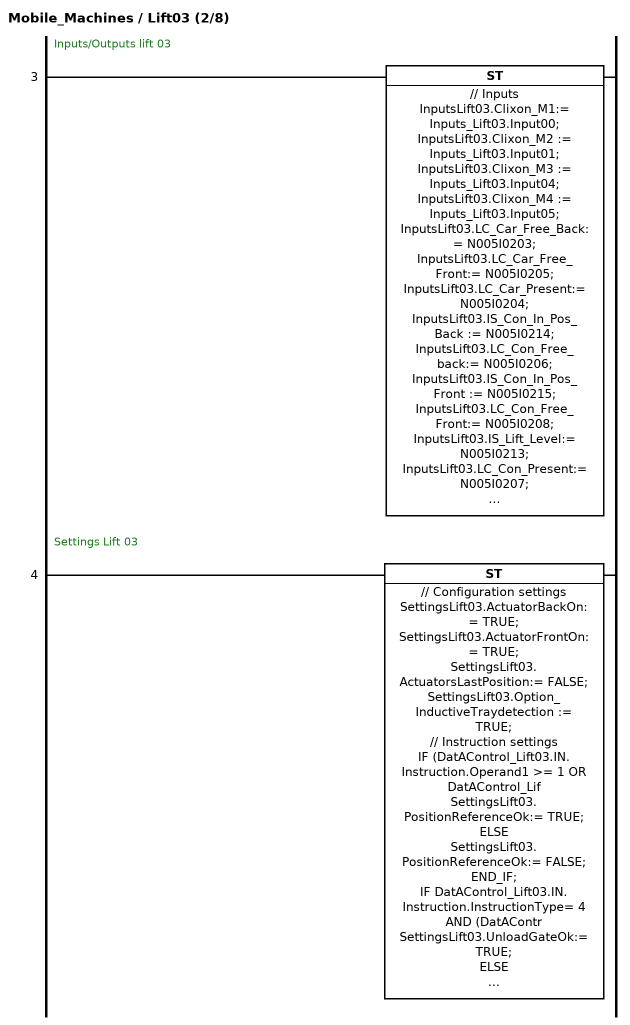
(* [picture p6: Mobile_Machines / Lift03, rungs 3-4] *)
(* Rung 3: Inputs/Outputs lift 03 *)
// Inputs
InputsLift03.Clixon_M1:= Inputs_Lift03.Input00;
InputsLift03.Clixon_M2 := Inputs_Lift03.Input01;
InputsLift03.Clixon_M3 := Inputs_Lift03.Input04;
InputsLift03.Clixon_M4 := Inputs_Lift03.Input05;
InputsLift03.LC_Car_Free_Back:= N005I0203;
InputsLift03.LC_Car_Free_Front:= N005I0205;
InputsLift03.LC_Car_Present:= N005I0204;
InputsLift03.IS_Con_In_Pos_Back := N005I0214;
InputsLift03.LC_Con_Free_back:= N005I0206;
InputsLift03.IS_Con_In_Pos_Front := N005I0215;
InputsLift03.LC_Con_Free_Front:= N005I0208;
InputsLift03.IS_Lift_Level:= N005I0213;
InputsLift03.LC_Con_Present:= N005I0207;
InputsLift03.LS_FallProtect:= N005I0200 OR TRUE;
InputsLift03.LS_Lift_Down:= N005I0202;
InputsLift03.LS_Lift_Up:= N005I0201;
InputsLift03.IS_Act_Back_In:= N005I0210; // Stopper blocks carrier
InputsLift03.IS_Act_Back_Out:= N005I0209; // Carrier can drive in
InputsLift03.IS_Act_Front_In:= N005I0212; // Stopper blocks carrier
InputsLift03.IS_Act_Front_Out:= N005I0211; // Carrier can drive in
InputsLift03.RC_Tray_Stopper_Min_Back_Up:= Inputs_Lift03_Ch.Input00;
InputsLift03.RC_Tray_Stopper_Max_Back_Up:= Inputs_Lift03_Ch.Input01;
InputsLift03.RC_Tray_Stopper_Min_Front_Up:= Inputs_Lift03_Ch.Input04;
InputsLift03.RC_Tray_Stopper_Max_Front_Up:= Inputs_Lift03_Ch.Input05;
InputsLift03.IO_OK := FALSE;
IF NOT N05_Major_Fault AND NOT N05_Minor_Fault AND NOT N05_Partial_Fault AND NOT N33_Major_Fault AND NOT N33_Minor_Fault AND NOT N33_Partial_Fault THEN
 InputsLift03.IO_OK := TRUE;
END_IF;

// Inputs rack
InputsLift03.LC_Lift_Free_Back[0]:= N005I0300;
InputsLift03.LC_Lift_Free_Back[1]:= TRUE;
InputsLift03.LC_Lift_Free_Back[2]:= TRUE;
InputsLift03.LC_Lift_Free_Back[3]:= TRUE;
InputsLift03.LC_Lift_Free_Back[4]:= N005I0304;
InputsLift03.LC_Lift_Free_Back[5]:= TRUE;
InputsLift03.LC_Lift_Free_Back[6]:= TRUE;
InputsLift03.LC_Lift_Free_Back[7]:= TRUE;
InputsLift03.LC_Lift_Free_Back[8]:= TRUE;
InputsLift03.LC_Lift_Free_Back[9]:= TRUE;
InputsLift03.LC_Lift_Free_Back[10]:= TRUE;
InputsLift03.LC_Lift_Free_Back[11]:= TRUE;
InputsLift03.LC_Lift_Free_Back[12]:= TRUE;
InputsLift03.LC_Lift_Free_Back[13]:= TRUE;
InputsLift03.LC_Lift_Free_Back[14]:= TRUE;
InputsLift03.LC_Lift_Free_Back[15]:= TRUE;

InputsLift03.LC_Lift_Free_Front[0]:= N005I0308;
InputsLift03.LC_Lift_Free_Front[1]:= N005I0309;
InputsLift03.LC_Lift_Free_Front[2]:= N005I0310;
InputsLift03.LC_Lift_Free_Front[3]:= N005I0311;
InputsLift03.LC_Lift_Free_Front[4]:= N005I0312;
InputsLift03.LC_Lift_Free_Front[5]:= N005I0313;
InputsLift03.LC_Lift_Free_Front[6]:= N005I0314;
InputsLift03.LC_Lift_Free_Front[7]:= N005I0315;
InputsLift03.LC_Lift_Free_Front[8]:= TRUE;
InputsLift03.LC_Lift_Free_Front[9]:= TRUE;
InputsLift03.LC_Lift_Free_Front[10]:= TRUE;
InputsLift03.LC_Lift_Free_Front[11]:= TRUE;
InputsLift03.LC_Lift_Free_Front[12]:= TRUE;
InputsLift03.LC_Lift_Free_Front[13]:= TRUE;
InputsLift03.LC_Lift_Free_Front[14]:= TRUE;
InputsLift03.LC_Lift_Free_Front[15]:= TRUE;

// Martins inputs
Lift03_SafetyInput1 := Inputs_Lift03.Input02;
Lift03_SafetyInput2 := Inputs_Lift03.Input03;

Knop_FW_Lift03 := N005I0301;
Knop_RV_Lift03 := N005I0302;
Knop_OK_Lift03 := N005I0303;
Knop_Snel_Lift03 := N005I0305;

// Outputs
N005O400:= OutputsLift03.Brake_Back;
// N005O401:= OutputsLift03.Actuator_Back_Out;
// N005O402:= OutputsLift03.Actuator_Back_In;
N005O403:= OutputsLift03.Actuator_Front_Out;
N005O404:= OutputsLift03.Actuator_Front_In;
N005O405 := OutputsLift03.Brake_Front; // Pls use only hold the brake and not release it for a correction
N005O406 := Led_RS_Extern;
N005O407 := OutputsLift03.V_TrayStopper_Front_Up;
LiftGR03NotLoaded := OutputsLift03.LC_Container_Free;

Comm_To_Carrier01.Lift_Info.CarrierNot_Loaded_Lift1 := FALSE; 
Comm_To_Carrier02.Lift_Info.CarrierNot_Loaded_Lift1 := FALSE;
Comm_To_Carrier03.Lift_Info.CarrierNot_Loaded_Lift1 := FALSE;
Comm_To_Carrier04.Lift_Info.CarrierNot_Loaded_Lift1 := FALSE;
Comm_To_Carrier05.Lift_Info.CarrierNot_Loaded_Lift1 := FALSE;

IF OutputsLift03.LC_Carrier_Free THEN
Comm_To_Carrier01.Lift_Info.CarrierNot_Loaded_Lift1 := TRUE; 
Comm_To_Carrier02.Lift_Info.CarrierNot_Loaded_Lift1 := TRUE;
Comm_To_Carrier03.Lift_Info.CarrierNot_Loaded_Lift1 := TRUE;
Comm_To_Carrier04.Lift_Info.CarrierNot_Loaded_Lift1 := TRUE;
Comm_To_Carrier05.Lift_Info.CarrierNot_Loaded_Lift1 := TRUE;
END_IF;

Comm_To_Carrier01.Lift_Info.TrayNot_Loaded_Lift1 := FALSE;
Comm_To_Carrier02.Lift_Info.TrayNot_Loaded_Lift1 := FALSE;
Comm_To_Carrier03.Lift_Info.TrayNot_Loaded_Lift1 := FALSE;
Comm_To_Carrier04.Lift_Info.TrayNot_Loaded_Lift1 := FALSE;
Comm_To_Carrier05.Lift_Info.TrayNot_Loaded_Lift1 := FALSE;

IF OutputsLift03.LC_Container_Free THEN
Comm_To_Carrier01.Lift_Info.TrayNot_Loaded_Lift1 := TRUE;
Comm_To_Carrier02.Lift_Info.TrayNot_Loaded_Lift1 := TRUE;
Comm_To_Carrier03.Lift_Info.TrayNot_Loaded_Lift1 := TRUE;
Comm_To_Carrier04.Lift_Info.TrayNot_Loaded_Lift1 := TRUE;
Comm_To_Carrier05.Lift_Info.TrayNot_Loaded_Lift1 := TRUE;
END_IF;
(* Rung 4: Settings Lift 03 *)
// Configuration settings
SettingsLift03.ActuatorBackOn:= TRUE;
SettingsLift03.ActuatorFrontOn:= TRUE;
SettingsLift03.ActuatorsLastPosition:= FALSE;
SettingsLift03.Option_InductiveTraydetection := TRUE;

// Instruction settings
IF (DatAControl_Lift03.IN.Instruction.Operand1 >= 1 OR DatAControl_Lift03.IN.Instruction.Operand1 <= 7) THEN
	SettingsLift03.PositionReferenceOk:= TRUE;
ELSE
	SettingsLift03.PositionReferenceOk:= FALSE;
END_IF;

IF DatAControl_Lift03.IN.Instruction.InstructionType= 4 AND (DatAControl_Lift03.IN.Instruction.Operand1 = 102 OR DatAControl_Lift03.IN.Instruction.Operand1 = 602) THEN
	SettingsLift03.UnloadGateOk:= TRUE;
ELSE
	SettingsLift03.UnloadGateOk:=FALSE;
END_IF;

IF DatAControl_Lift03.IN.Instruction.InstructionType= 3 AND (DatAControl_Lift03.IN.Instruction.Operand1 = 102 OR DatAControl_Lift03.IN.Instruction.Operand1 = 602) THEN
	SettingsLift03.LoadGateOk:= TRUE;
ELSE
	SettingsLift03.LoadGateOk:= FALSE;
END_IF;

// Parameters
SettingsLift03.MachineCode:=4;
SettingsLift03.SafeStopTime:=15;
SettingsLift03.Tolerance_At_Position:=50;
SettingsLift03.Warning_Tolerance_At_Position:=25;
SettingsLift03.BrakeReleaseFreq:=750;
SettingsLift03.Dec_Area_High:= 10000;
SettingsLift03.Dec_Area_Low:=1000;
SettingsLift03.NodeNummerLift:=9;
SettingsLift03.NodeNummerChain:=10;
SettingsLift03.MinimumSpeed:=1000;
SettingsLift03.MaximumSpeed:=8400; // Motor with extern brake 84Hz max, motor with no brake 87Hz max
SettingsLift03.MinimumSpeedChain:= 3700;
SettingsLift03.MaximumSpeedChain:= 8000; // Motor with intern brake 68 Hz max
SettingsLift03.TimeConFreeBackDOFF:= 50;
SettingsLift03.TimeConFreeBackDON:= 5;
SettingsLift03.TimeConFreeFrontDOFF:= 5;
SettingsLift03.TimeConFreeFrontDON:= 5;
SettingsLift03.UseBenchUnloadInstruction:= TRUE;

IF Commands_Lift03.Reverse THEN // Slow down
	SettingsLift03.MinimumSpeed := 750;
	SettingsLift03.BrakeReleaseFreq:=500;
END_IF;

IF SettingsLift03.Option_InductiveTraydetection THEN
	SettingsLift03.ChainHighSpeed := 60;
ELSE
 	SettingsLift03.ChainHighSpeed := 85;
END_IF;

SettingsLift03.TimeConInductiveBackDOFF := 2;
SettingsLift03.TimeConInductiveBackDON := 8;
SettingsLift03.TimeConInductiveFrontDOFF := 2;
SettingsLift03.TimeConInductiveFrontDON := 8;

// Mechanical settings 1mm = 17 pulses
SettingsLift03.MinimumPulseLevel:=10000;
SettingsLift03.MaximumPulseLevel:=177000;
SettingsLift03.TooFarAllowed:= 1000;
SettingsLift03.ResetValueMargin := 500;
SettingsLift03.MinimumPosition:= 1;
SettingsLift03.MaximumPosition:= 9;
SettingsLift03.PulseLevel[1]:=10000;
SettingsLift03.PulseLevel[2]:= Lift3_PulsValueLevel2; // 13345;
SettingsLift03.PulseLevel[3]:= Lift3_PulsValueLevel3; // 49853 // 49790
SettingsLift03.PulseLevel[4]:= Lift3_PulsValueLevel4; // 70329 // 70240; 
SettingsLift03.PulseLevel[5]:= Lift3_PulsValueLevel5; // 90761 // 90690; 
SettingsLift03.PulseLevel[6]:= Lift3_PulsValueLevel6; // 111397 // 111140; 
SettingsLift03.PulseLevel[7]:= Lift3_PulsValueLevel7; // 131690 // 131590;
SettingsLift03.PulseLevel[8]:= Lift3_PulsValueLevel8; // 152156 // 152040; 
SettingsLift03.PulseLevel[9]:= Lift3_PulsValueLevel9; // 172626 // 172490; 
SettingsLift03.PulseLevel[10]:=10;
SettingsLift03.PulseLevel[11]:=10;
SettingsLift03.PulseLevel[12]:=10;
SettingsLift03.PulseLevel[13]:=10;
SettingsLift03.PulseLevel[14]:=10;
SettingsLift03.PulseLevel[15]:=10;

SettingsLift03.NeedLevelSensor[1]:=FALSE;
SettingsLift03.NeedLevelSensor[2]:=FALSE;
SettingsLift03.NeedLevelSensor[3]:=TRUE;
SettingsLift03.NeedLevelSensor[4]:=TRUE;
SettingsLift03.NeedLevelSensor[5]:=TRUE;
SettingsLift03.NeedLevelSensor[6]:=TRUE;
SettingsLift03.NeedLevelSensor[7]:=TRUE;
SettingsLift03.NeedLevelSensor[8]:=TRUE;
SettingsLift03.NeedLevelSensor[9]:=TRUE;
SettingsLift03.NeedLevelSensor[10]:=TRUE;
SettingsLift03.NeedLevelSensor[11]:=TRUE;
SettingsLift03.NeedLevelSensor[12]:=TRUE;
SettingsLift03.NeedLevelSensor[13]:=TRUE;
SettingsLift03.NeedLevelSensor[14]:=TRUE;
SettingsLift03.NeedLevelSensor[15]:=TRUE;

// SettingsLift03.BrakeReleaseFreq:=750; SettingsLift03.MinimumSpeed:=1000;
// When rev setting: SettingsLift03.MinimumSpeed := 750; SettingsLift03.BrakeReleaseFreq:=500;
// Acc 20sec, dec 4sec

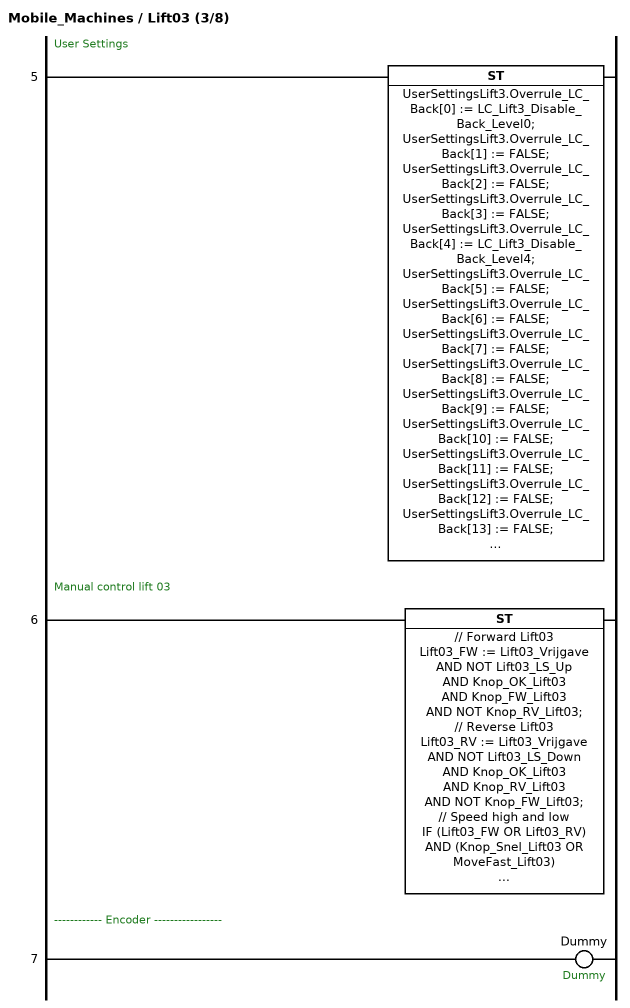
(* Rung 5: User Settings *)
UserSettingsLift3.Overrule_LC_Back[0] := LC_Lift3_Disable_Back_Level0;
UserSettingsLift3.Overrule_LC_Back[1] := FALSE;
UserSettingsLift3.Overrule_LC_Back[2] := FALSE;
UserSettingsLift3.Overrule_LC_Back[3] := FALSE;
UserSettingsLift3.Overrule_LC_Back[4] := LC_Lift3_Disable_Back_Level4;
UserSettingsLift3.Overrule_LC_Back[5] := FALSE;
UserSettingsLift3.Overrule_LC_Back[6] := FALSE;
UserSettingsLift3.Overrule_LC_Back[7] := FALSE;
UserSettingsLift3.Overrule_LC_Back[8] := FALSE;
UserSettingsLift3.Overrule_LC_Back[9] := FALSE;
UserSettingsLift3.Overrule_LC_Back[10] := FALSE;
UserSettingsLift3.Overrule_LC_Back[11] := FALSE;
UserSettingsLift3.Overrule_LC_Back[12] := FALSE;
UserSettingsLift3.Overrule_LC_Back[13] := FALSE;
UserSettingsLift3.Overrule_LC_Back[14] := FALSE;
UserSettingsLift3.Overrule_LC_Back[15] := FALSE;

UserSettingsLift3.Overrule_LC_Front[0] := LC_Lift3_Disable_Front_Level0;
UserSettingsLift3.Overrule_LC_Front[1] := LC_Lift3_Disable_Front_Level1;
UserSettingsLift3.Overrule_LC_Front[2] := LC_Lift3_Disable_Front_Level2;
UserSettingsLift3.Overrule_LC_Front[3] := LC_Lift3_Disable_Front_Level3;
UserSettingsLift3.Overrule_LC_Front[4] := LC_Lift3_Disable_Front_Level4;
UserSettingsLift3.Overrule_LC_Front[5] := LC_Lift3_Disable_Front_Level5;
UserSettingsLift3.Overrule_LC_Front[6] := LC_Lift3_Disable_Front_Level6;
UserSettingsLift3.Overrule_LC_Front[7] := LC_Lift3_Disable_Front_Level7;
UserSettingsLift3.Overrule_LC_Front[8] := FALSE;
UserSettingsLift3.Overrule_LC_Front[9] := FALSE;
UserSettingsLift3.Overrule_LC_Front[10] := FALSE;
UserSettingsLift3.Overrule_LC_Front[11] := FALSE;
UserSettingsLift3.Overrule_LC_Front[12] := FALSE;
UserSettingsLift3.Overrule_LC_Front[13] := FALSE;
UserSettingsLift3.Overrule_LC_Front[14] := FALSE;
UserSettingsLift3.Overrule_LC_Front[15] := FALSE;
(* Rung 6: Manual control lift 03 *)
// Forward Lift03
Lift03_FW := Lift03_Vrijgave
AND NOT Lift03_LS_Up
AND Knop_OK_Lift03
AND Knop_FW_Lift03
AND NOT Knop_RV_Lift03;
// Reverse Lift03
Lift03_RV := Lift03_Vrijgave
AND NOT Lift03_LS_Down
AND Knop_OK_Lift03
AND Knop_RV_Lift03
AND NOT Knop_FW_Lift03;

// Speed high and low
IF (Lift03_FW OR Lift03_RV) AND (Knop_Snel_Lift03 OR MoveFast_Lift03)
AND EncoderLift03>SettingsLift03.MinimumPulseLevel+1000 AND EncoderLift03<SettingsLift03.MaximumPulseLevel-1000 THEN
	SettingsLift03.MinimumSpeed:=5000;
END_IF;

// Led ok Lift03
Led_Knop_OK_Lift03 := Knop_OK_Lift03 AND Lift03_Vrijgave;

// Vrijgave Lift03
Lift03_Vrijgave := (*Lift03_LS_FallProtect
AND*) Lift03_SafetyInput1 AND Lift03_SafetyInput2 AND Lift03_Alarms=0;

// Use manual control buttons as replacement for pocket (TEMP)
//Lift03_FW  Lift03_RV
IF Knop_OK_Lift03 THEN
	Pocket_Lift03.Move.Out:=Lift03_FW;
	Pocket_Lift03.Move.In:= Lift03_RV;
	Pocket_Lift03.Move.Stop:= NOT Lift03_FW AND NOT Lift03_RV;
END_IF;

// Move fast on/off
IF Pocket_Lift03.MoveFastOn THEN
	MoveFast_Lift03 := TRUE;
END_IF;
IF Pocket_Lift03.MoveFastOff OR DatAControl_Lift03.IN.MachineMode<>3 THEN
	MoveFast_Lift03 := FALSE;
END_IF;
Pocket_Lift03.MoveFastOn := FALSE;
Pocket_Lift03.MoveFastOff := FALSE;
(* Rung 7: ------------ Encoder ----------------- *)
Dummy := TRUE;

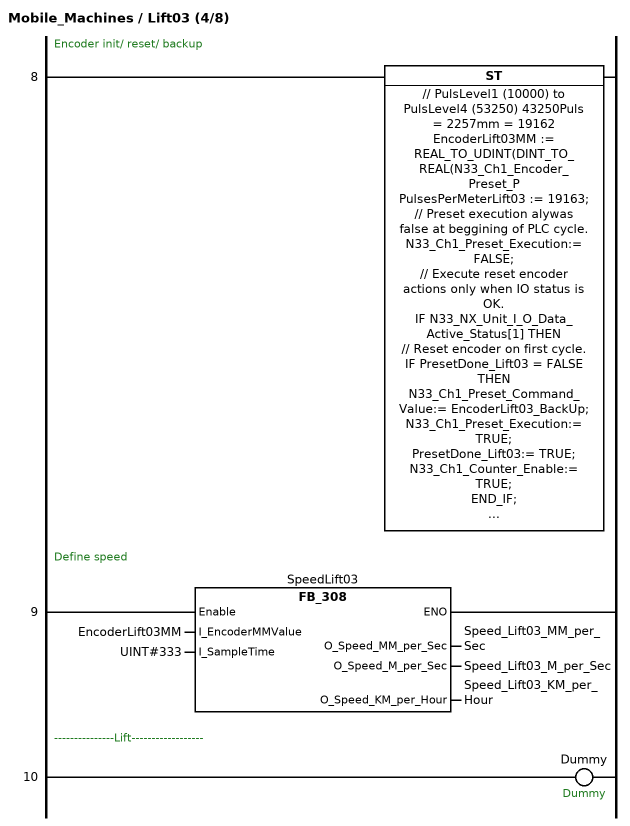
(* Rung 8: Encoder init/ reset/ backup *)
// PulsLevel1 (10000) to PulsLevel4 (53250) 43250Puls = 2257mm = 19162,605228179 PpM
EncoderLift03MM := REAL_TO_UDINT(DINT_TO_REAL(N33_Ch1_Encoder_Preset_Position) / UDINT_TO_REAL(PulsesPerMeterLift03) * 1000);
PulsesPerMeterLift03 := 19163;

// Preset execution alywas false at beggining of PLC cycle.
N33_Ch1_Preset_Execution:= FALSE;

// Execute reset encoder actions only when IO status is OK.
IF N33_NX_Unit_I_O_Data_Active_Status[1] THEN
	
	// Reset encoder on first cycle.
	IF PresetDone_Lift03 = FALSE THEN
		N33_Ch1_Preset_Command_Value:= EncoderLift03_BackUp;
		N33_Ch1_Preset_Execution:= TRUE;
		PresetDone_Lift03:= TRUE;
		N33_Ch1_Counter_Enable:= TRUE;
	END_IF;
	
	// Reset encoder when lift is at position.
	IF ResetEncoder_Lift03 THEN
		N33_Ch1_Preset_Command_Value:= ResetEncoderValue_Lift03; // 10000 @Ground
		N33_Ch1_Preset_Execution:= TRUE;
		ResetEncoder_Lift03:= FALSE;
	END_IF;
	
	// Move encoder value.
    EncoderLift03 := DINT_TO_UDINT(N33_Ch1_Encoder_Preset_Position);
		
	// Backup encoder value.
	EncoderLift03_Backup:= EncoderLift03;
END_IF;
(* Rung 9: Define speed *)
SpeedLift03(Enable := TRUE, I_EncoderMMValue := EncoderLift03MM, I_SampleTime := UINT#333, O_Speed_MM_per_Sec => Speed_Lift03_MM_per_Sec, O_Speed_M_per_Sec => Speed_Lift03_M_per_Sec, O_Speed_KM_per_Hour => Speed_Lift03_KM_per_Hour);
(* Rung 10: ---------------Lift------------------ *)
Dummy := TRUE;

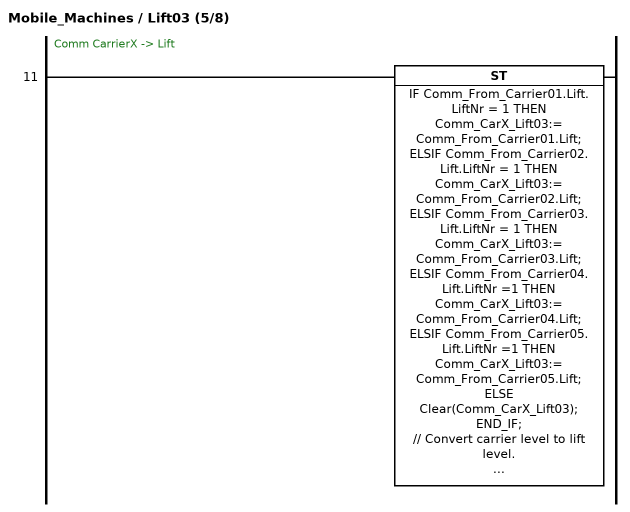
(* Rung 11: Comm CarrierX -> Lift *)
IF Comm_From_Carrier01.Lift.LiftNr = 1 THEN
	Comm_CarX_Lift03:= Comm_From_Carrier01.Lift;
ELSIF Comm_From_Carrier02.Lift.LiftNr = 1 THEN
	Comm_CarX_Lift03:= Comm_From_Carrier02.Lift;
ELSIF Comm_From_Carrier03.Lift.LiftNr = 1 THEN
	Comm_CarX_Lift03:= Comm_From_Carrier03.Lift;
ELSIF Comm_From_Carrier04.Lift.LiftNr =1 THEN
	Comm_CarX_Lift03:= Comm_From_Carrier04.Lift;
ELSIF Comm_From_Carrier05.Lift.LiftNr =1 THEN
	Comm_CarX_Lift03:= Comm_From_Carrier05.Lift;
ELSE
	Clear(Comm_CarX_Lift03);
END_IF;

// Convert carrier level to lift level.
//This is only needed when lift has more levels than the carrier!
CASE Comm_CarX_Lift03.Height_MobileMachine OF
	1: Comm_CarX_Lift03.Height_MobileMachine:=3;
	2: Comm_CarX_Lift03.Height_MobileMachine:=4;
	// mezzanine will probably add an extra level to the lift ones.
	3: Comm_CarX_Lift03.Height_MobileMachine:=5;
	4: Comm_CarX_Lift03.Height_MobileMachine:=6;
	5: Comm_CarX_Lift03.Height_MobileMachine:=7;
	6: Comm_CarX_Lift03.Height_MobileMachine:=8;
	7: Comm_CarX_Lift03.Height_MobileMachine:=9;
ELSE
	// If lift drops the carrier on a level not listed above set to 0 to avoid wrong positions.
     Comm_CarX_Lift03.Height_MobileMachine:=0;
END_CASE;

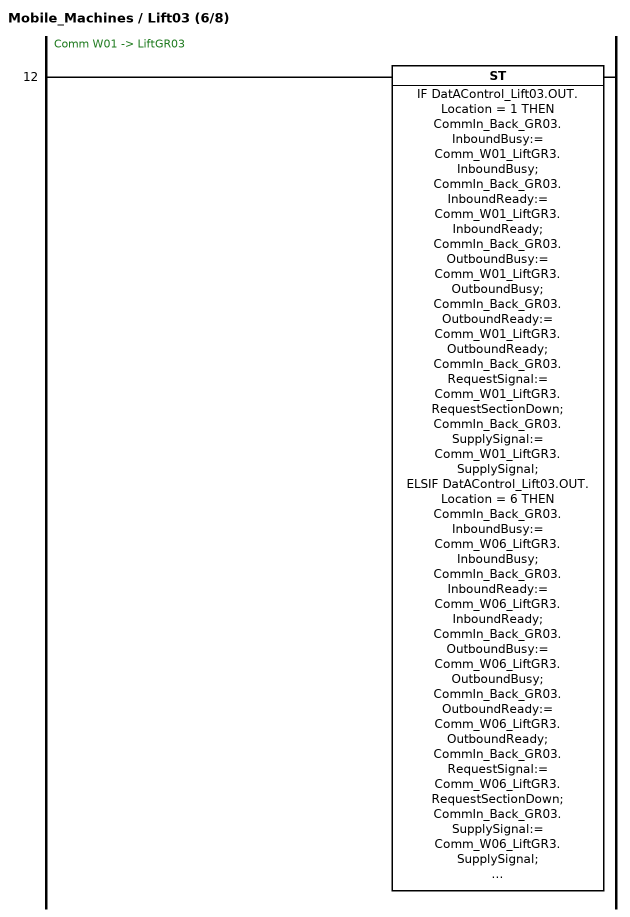
(* Rung 12: Comm W01 -> LiftGR03 *)
IF DatAControl_Lift03.OUT.Location = 1 THEN
CommIn_Back_GR03.InboundBusy:= Comm_W01_LiftGR3.InboundBusy;
CommIn_Back_GR03.InboundReady:= Comm_W01_LiftGR3.InboundReady;
CommIn_Back_GR03.OutboundBusy:= Comm_W01_LiftGR3.OutboundBusy;
CommIn_Back_GR03.OutboundReady:= Comm_W01_LiftGR3.OutboundReady;
CommIn_Back_GR03.RequestSignal:= Comm_W01_LiftGR3.RequestSectionDown;
CommIn_Back_GR03.SupplySignal:= Comm_W01_LiftGR3.SupplySignal;
ELSIF DatAControl_Lift03.OUT.Location = 6 THEN
CommIn_Back_GR03.InboundBusy:= Comm_W06_LiftGR3.InboundBusy;
CommIn_Back_GR03.InboundReady:= Comm_W06_LiftGR3.InboundReady;
CommIn_Back_GR03.OutboundBusy:= Comm_W06_LiftGR3.OutboundBusy;
CommIn_Back_GR03.OutboundReady:= Comm_W06_LiftGR3.OutboundReady;
CommIn_Back_GR03.RequestSignal:= Comm_W06_LiftGR3.RequestSectionDown;
CommIn_Back_GR03.SupplySignal:= Comm_W06_LiftGR3.SupplySignal;
END_IF;

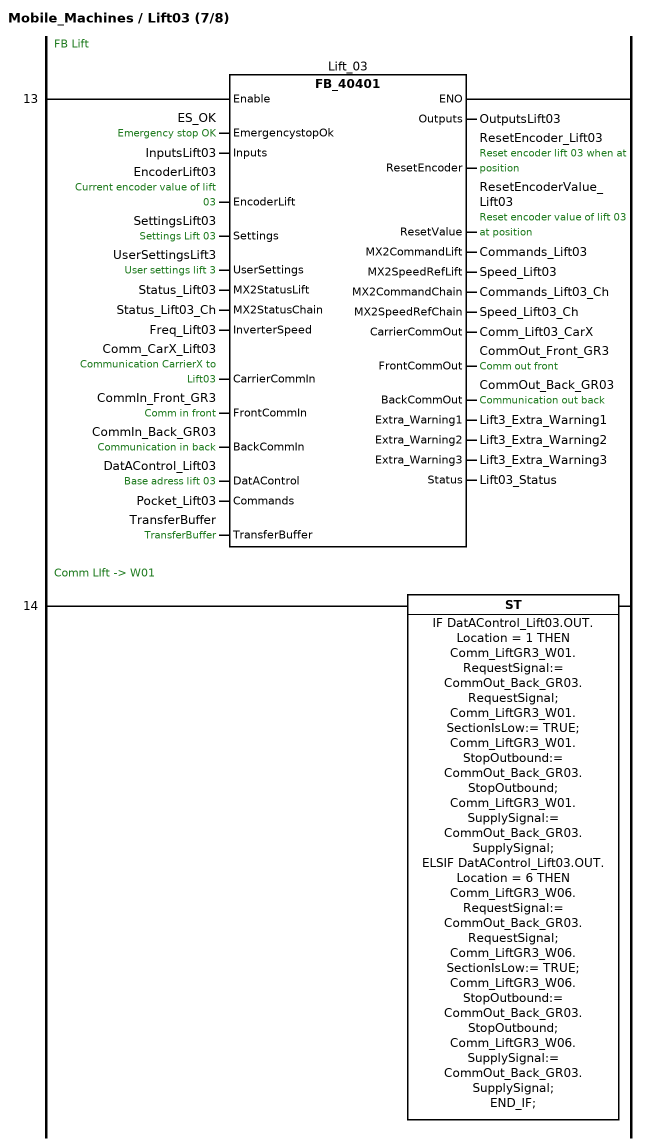
(* Rung 13: FB Lift *)
Lift_03(Enable := TRUE, EmergencystopOk := ES_OK, Inputs := InputsLift03, EncoderLift := EncoderLift03, Settings := SettingsLift03, UserSettings := UserSettingsLift3, MX2StatusLift := Status_Lift03, MX2StatusChain := Status_Lift03_Ch, InverterSpeed := Freq_Lift03, CarrierCommIn := Comm_CarX_Lift03, FrontCommIn := CommIn_Front_GR3, BackCommIn := CommIn_Back_GR03, DatAControl := DatAControl_Lift03, Commands := Pocket_Lift03, TransferBuffer := TransferBuffer, Outputs => OutputsLift03, ResetEncoder => ResetEncoder_Lift03, ResetValue => ResetEncoderValue_Lift03, MX2CommandLift => Commands_Lift03, MX2SpeedRefLift => Speed_Lift03, MX2CommandChain => Commands_Lift03_Ch, MX2SpeedRefChain => Speed_Lift03_Ch, CarrierCommOut => Comm_Lift03_CarX, FrontCommOut => CommOut_Front_GR3, BackCommOut => CommOut_Back_GR03, Extra_Warning1 => Lift3_Extra_Warning1, Extra_Warning2 => Lift3_Extra_Warning2, Extra_Warning3 => Lift3_Extra_Warning3, Status => Lift03_Status);
(* Rung 14: Comm LIft -> W01 *)
IF DatAControl_Lift03.OUT.Location = 1 THEN
Comm_LiftGR3_W01.RequestSignal:= CommOut_Back_GR03.RequestSignal;
Comm_LiftGR3_W01.SectionIsLow:= TRUE;
Comm_LiftGR3_W01.StopOutbound:= CommOut_Back_GR03.StopOutbound;
Comm_LiftGR3_W01.SupplySignal:= CommOut_Back_GR03.SupplySignal;
ELSIF DatAControl_Lift03.OUT.Location = 6 THEN
Comm_LiftGR3_W06.RequestSignal:= CommOut_Back_GR03.RequestSignal;
Comm_LiftGR3_W06.SectionIsLow:= TRUE;
Comm_LiftGR3_W06.StopOutbound:= CommOut_Back_GR03.StopOutbound;
Comm_LiftGR3_W06.SupplySignal:= CommOut_Back_GR03.SupplySignal;
END_IF;

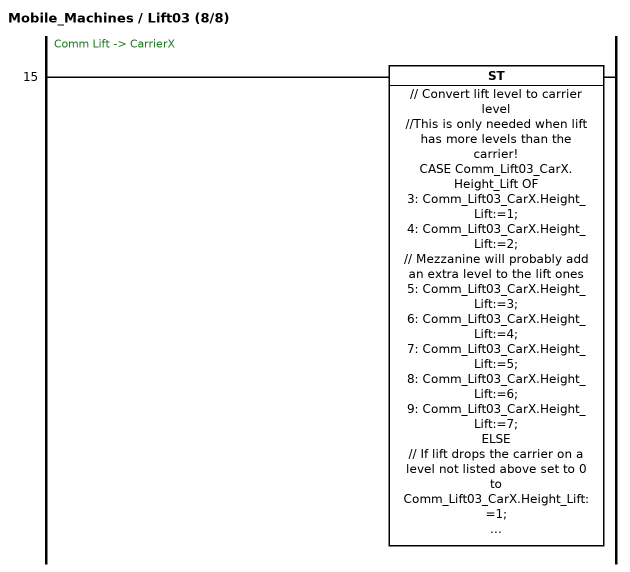
(* Rung 15: Comm Lift -> CarrierX *)
// Convert lift level to carrier level
//This is only needed when lift has more levels than the carrier!
CASE Comm_Lift03_CarX.Height_Lift OF
	3: Comm_Lift03_CarX.Height_Lift:=1;
	4: Comm_Lift03_CarX.Height_Lift:=2;
	// Mezzanine will probably add an extra level to the lift ones
	5: Comm_Lift03_CarX.Height_Lift:=3;
	6: Comm_Lift03_CarX.Height_Lift:=4;
	7: Comm_Lift03_CarX.Height_Lift:=5;
	8: Comm_Lift03_CarX.Height_Lift:=6;
	9: Comm_Lift03_CarX.Height_Lift:=7;
ELSE
	// If lift drops the carrier on a level not listed above set to 0 to avoid wrong positions.
     Comm_Lift03_CarX.Height_Lift:=1;
END_CASE;

IF Comm_From_Carrier01.Lift.LiftNr = 1 THEN
	Comm_To_Carrier01.Lift:= Comm_Lift03_CarX;
ELSIF Comm_From_Carrier02.Lift.LiftNr = 1 THEN
	Comm_To_Carrier02.Lift:= Comm_Lift03_CarX;
ELSIF Comm_From_Carrier03.Lift.LiftNr = 1 THEN
	Comm_To_Carrier03.Lift:= Comm_Lift03_CarX;
ELSIF Comm_From_Carrier04.Lift.LiftNr = 1 THEN
	Comm_To_Carrier04.Lift:= Comm_Lift03_CarX;
ELSIF Comm_From_Carrier05.Lift.LiftNr = 1 THEN
	Comm_To_Carrier05.Lift:= Comm_Lift03_CarX;
END_IF;

(* Section Lift04: ladder, written here as Structured Text *)

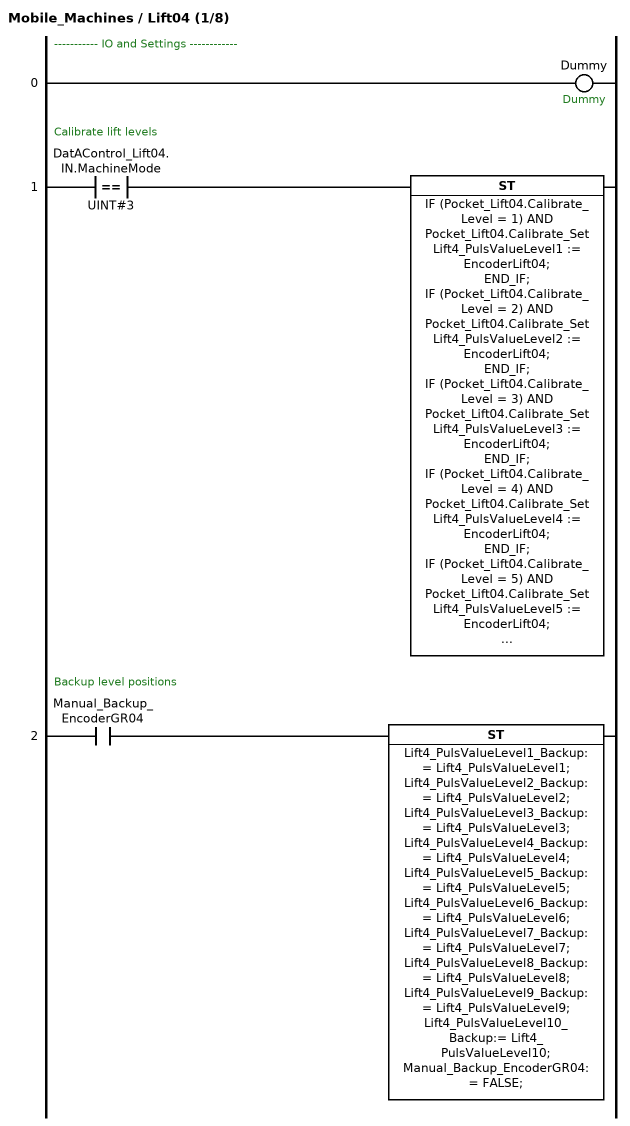
(* Rung 0: ----------- IO and Settings ------------ *)
Dummy := TRUE;
(* Rung 1: Calibrate lift levels *)
IF DatAControl_Lift04.IN.MachineMode = UINT#3 THEN
    IF (Pocket_Lift04.Calibrate_Level = 1) AND Pocket_Lift04.Calibrate_SetLevel THEN
    	Lift4_PulsValueLevel1 := EncoderLift04;
    END_IF;
    
    IF (Pocket_Lift04.Calibrate_Level = 2) AND Pocket_Lift04.Calibrate_SetLevel THEN
    	Lift4_PulsValueLevel2 := EncoderLift04;
    END_IF;
    
    IF (Pocket_Lift04.Calibrate_Level = 3) AND Pocket_Lift04.Calibrate_SetLevel THEN
    	Lift4_PulsValueLevel3 := EncoderLift04;
    END_IF;
    
    IF (Pocket_Lift04.Calibrate_Level = 4) AND Pocket_Lift04.Calibrate_SetLevel THEN
    	Lift4_PulsValueLevel4 := EncoderLift04;
    END_IF;
    
    IF (Pocket_Lift04.Calibrate_Level = 5) AND Pocket_Lift04.Calibrate_SetLevel THEN
    	Lift4_PulsValueLevel5 := EncoderLift04;
    END_IF;
    
    IF (Pocket_Lift04.Calibrate_Level = 6) AND Pocket_Lift04.Calibrate_SetLevel THEN
    	Lift4_PulsValueLevel6 := EncoderLift04;
    END_IF;
    
    IF (Pocket_Lift04.Calibrate_Level = 7) AND Pocket_Lift04.Calibrate_SetLevel THEN
    	Lift4_PulsValueLevel7 := EncoderLift04;
    END_IF;
    
    IF (Pocket_Lift04.Calibrate_Level = 8) AND Pocket_Lift04.Calibrate_SetLevel THEN
    	Lift4_PulsValueLevel8 := EncoderLift04;
    END_IF;
    
    IF (Pocket_Lift04.Calibrate_Level = 9) AND Pocket_Lift04.Calibrate_SetLevel THEN
    	Lift4_PulsValueLevel9 := EncoderLift04;
    END_IF;
    
    IF (Pocket_Lift04.Calibrate_Level = 10) AND Pocket_Lift04.Calibrate_SetLevel THEN
    	Lift4_PulsValueLevel10 := EncoderLift04;
    END_IF;
    
    Pocket_Lift04.Calibrate_SetLevel := FALSE; 
END_IF;
(* Rung 2: Backup level positions *)
IF Manual_Backup_EncoderGR04 THEN
    Lift4_PulsValueLevel1_Backup:= Lift4_PulsValueLevel1;
    Lift4_PulsValueLevel2_Backup:= Lift4_PulsValueLevel2;
    Lift4_PulsValueLevel3_Backup:= Lift4_PulsValueLevel3;
    Lift4_PulsValueLevel4_Backup:= Lift4_PulsValueLevel4;
    Lift4_PulsValueLevel5_Backup:= Lift4_PulsValueLevel5;
    Lift4_PulsValueLevel6_Backup:= Lift4_PulsValueLevel6;
    Lift4_PulsValueLevel7_Backup:= Lift4_PulsValueLevel7;
    Lift4_PulsValueLevel8_Backup:= Lift4_PulsValueLevel8;
    Lift4_PulsValueLevel9_Backup:= Lift4_PulsValueLevel9;
    Lift4_PulsValueLevel10_Backup:= Lift4_PulsValueLevel10;
    
    Manual_Backup_EncoderGR04:= FALSE;
END_IF;

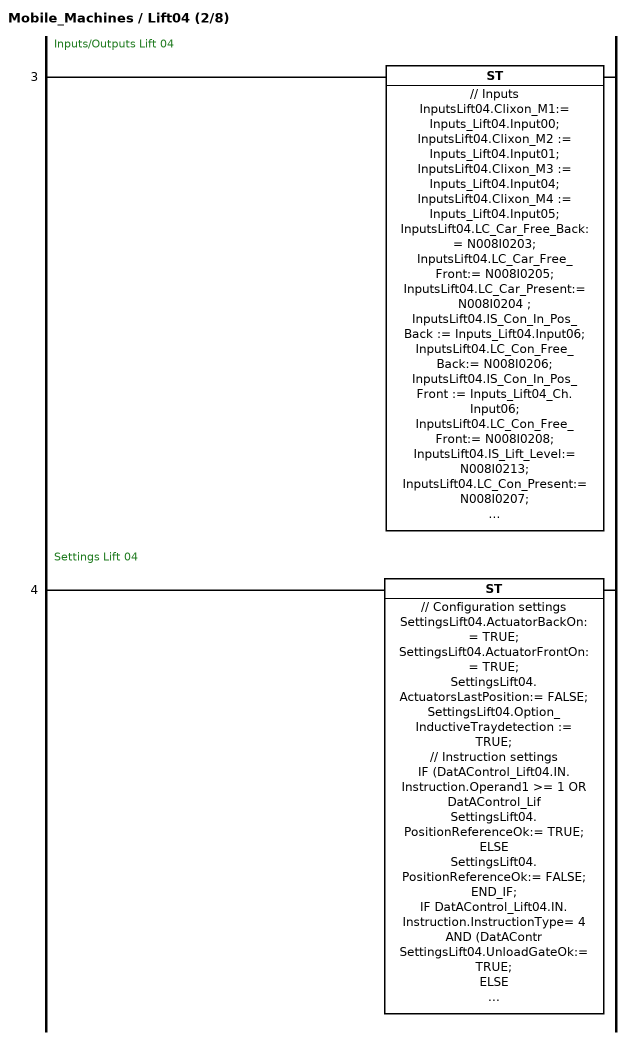
(* Rung 3: Inputs/Outputs Lift 04 *)
// Inputs
InputsLift04.Clixon_M1:= Inputs_Lift04.Input00;
InputsLift04.Clixon_M2 := Inputs_Lift04.Input01;
InputsLift04.Clixon_M3 := Inputs_Lift04.Input04;
InputsLift04.Clixon_M4 := Inputs_Lift04.Input05;
InputsLift04.LC_Car_Free_Back:= N008I0203;
InputsLift04.LC_Car_Free_Front:= N008I0205;
InputsLift04.LC_Car_Present:= N008I0204 ;
InputsLift04.IS_Con_In_Pos_Back := Inputs_Lift04.Input06;
InputsLift04.LC_Con_Free_Back:= N008I0206;
InputsLift04.IS_Con_In_Pos_Front := Inputs_Lift04_Ch.Input06;
InputsLift04.LC_Con_Free_Front:= N008I0208;
InputsLift04.IS_Lift_Level:= N008I0213;
InputsLift04.LC_Con_Present:= N008I0207;
InputsLift04.LS_FallProtect:= N008I0200;
InputsLift04.LS_Lift_Down:= N008I0202;
InputsLift04.LS_Lift_Up:= N008I0201;
InputsLift04.IS_Act_Back_In:= N008I0210; // Stopper blocks carrier
InputsLift04.IS_Act_Back_Out:= N008I0209; // Carrier can drive in
InputsLift04.IS_Act_Front_In:= N008I0212; // Stopper blocks carrier
InputsLift04.IS_Act_Front_Out:= N008I0211; // Carrier can drive in
InputsLift04.RC_Tray_Stopper_Min_Back_Up:= Inputs_Lift04_Ch.Input00;
InputsLift04.RC_Tray_Stopper_Max_Back_Up:= Inputs_Lift04_Ch.Input01;
InputsLift04.RC_Tray_Stopper_Min_Front_Up:= Inputs_Lift04_Ch.Input04;
InputsLift04.RC_Tray_Stopper_Max_Front_Up:= Inputs_Lift04_Ch.Input05;
InputsLift04.IO_OK := FALSE;
IF NOT N08_Major_Fault AND NOT N08_Minor_Fault AND NOT N08_Partial_Fault AND NOT N43_Major_Fault AND NOT N43_Minor_Fault AND NOT N43_Partial_Fault THEN
 InputsLift04.IO_OK := TRUE;
END_IF;

// Inputs rack
InputsLift04.LC_Lift_Free_Back[0]:= N008I0300;
InputsLift04.LC_Lift_Free_Back[1]:= TRUE;
InputsLift04.LC_Lift_Free_Back[2]:= TRUE;
InputsLift04.LC_Lift_Free_Back[3]:= TRUE;
InputsLift04.LC_Lift_Free_Back[4]:= N008I0304;
InputsLift04.LC_Lift_Free_Back[5]:= TRUE;
InputsLift04.LC_Lift_Free_Back[6]:= TRUE;
InputsLift04.LC_Lift_Free_Back[7]:= TRUE;
InputsLift04.LC_Lift_Free_Back[8]:= TRUE;
InputsLift04.LC_Lift_Free_Back[9]:= TRUE;
InputsLift04.LC_Lift_Free_Back[10]:= TRUE;
InputsLift04.LC_Lift_Free_Back[11]:= TRUE;
InputsLift04.LC_Lift_Free_Back[12]:= TRUE;
InputsLift04.LC_Lift_Free_Back[13]:= TRUE;
InputsLift04.LC_Lift_Free_Back[14]:= TRUE;
InputsLift04.LC_Lift_Free_Back[15]:= TRUE;

InputsLift04.LC_Lift_Free_Front[0]:= N008I0308;
InputsLift04.LC_Lift_Free_Front[1]:= N008I0309;
InputsLift04.LC_Lift_Free_Front[2]:= N008I0310;
InputsLift04.LC_Lift_Free_Front[3]:= N008I0311;
InputsLift04.LC_Lift_Free_Front[4]:= N008I0312;
InputsLift04.LC_Lift_Free_Front[5]:= N008I0313;
InputsLift04.LC_Lift_Free_Front[6]:= N008I0314;
InputsLift04.LC_Lift_Free_Front[7]:= N008I0315;
InputsLift04.LC_Lift_Free_Front[8]:= TRUE;
InputsLift04.LC_Lift_Free_Front[9]:= TRUE;
InputsLift04.LC_Lift_Free_Front[10]:= TRUE;
InputsLift04.LC_Lift_Free_Front[11]:= TRUE;
InputsLift04.LC_Lift_Free_Front[12]:= TRUE;
InputsLift04.LC_Lift_Free_Front[13]:= TRUE;
InputsLift04.LC_Lift_Free_Front[14]:= TRUE;
InputsLift04.LC_Lift_Free_Front[15]:= TRUE;

// Martins inputs
Lift04_SafetyInput1:= Inputs_Lift04.Input02;
Lift04_SafetyInput2:= Inputs_Lift04.Input03;

Knop_FW_Lift04:= N008I0301;
Knop_RV_Lift04:= N008I0302;
Knop_OK_Lift04:= N008I0303;
Knop_Snel_Lift04:= N008I0305;

// Outputs
N008O0400:= OutputsLift04.Brake_Back;
// N008O0401:= OutputsLift04.Actuator_Back_Out; THIS OUTPUT HAS BEEN REWIRED TO POWER CHARGER 3D105
// N008O0402:= OutputsLift04.Actuator_Back_In;
N008O0403:= OutputsLift04.Actuator_Front_Out;
N008O0404:= OutputsLift04.Actuator_Front_In;
N008O0405:= OutputsLift04.Brake_Front; // Pls use only hold the brake and not release it for a correction
N008O0406:= OutputsLift04.V_Traystopper_Back_Up;
N008O0407 := OutputsLift04.V_TrayStopper_Front_Up;
LiftGR04NotLoaded := OutputsLift04.LC_Container_Free;

Comm_To_Carrier01.Lift_Info.CarrierNot_Loaded_Lift2 := FALSE; 
Comm_To_Carrier02.Lift_Info.CarrierNot_Loaded_Lift2 := FALSE;
Comm_To_Carrier03.Lift_Info.CarrierNot_Loaded_Lift2 := FALSE;
Comm_To_Carrier04.Lift_Info.CarrierNot_Loaded_Lift2 := FALSE;
Comm_To_Carrier05.Lift_Info.CarrierNot_Loaded_Lift2 := FALSE;

IF OutputsLift04.LC_Carrier_Free THEN
Comm_To_Carrier01.Lift_Info.CarrierNot_Loaded_Lift2 := TRUE; 
Comm_To_Carrier02.Lift_Info.CarrierNot_Loaded_Lift2 := TRUE;
Comm_To_Carrier03.Lift_Info.CarrierNot_Loaded_Lift2 := TRUE;
Comm_To_Carrier04.Lift_Info.CarrierNot_Loaded_Lift2 := TRUE;
Comm_To_Carrier05.Lift_Info.CarrierNot_Loaded_Lift2 := TRUE;
END_IF;

Comm_To_Carrier01.Lift_Info.TrayNot_Loaded_Lift2 := FALSE;
Comm_To_Carrier02.Lift_Info.TrayNot_Loaded_Lift2 := FALSE;
Comm_To_Carrier03.Lift_Info.TrayNot_Loaded_Lift2 := FALSE;
Comm_To_Carrier04.Lift_Info.TrayNot_Loaded_Lift2 := FALSE;
Comm_To_Carrier05.Lift_Info.TrayNot_Loaded_Lift2 := FALSE;

IF OutputsLift04.LC_Container_Free THEN
Comm_To_Carrier01.Lift_Info.TrayNot_Loaded_Lift2 := TRUE;
Comm_To_Carrier02.Lift_Info.TrayNot_Loaded_Lift2 := TRUE;
Comm_To_Carrier03.Lift_Info.TrayNot_Loaded_Lift2 := TRUE;
Comm_To_Carrier04.Lift_Info.TrayNot_Loaded_Lift2 := TRUE;
Comm_To_Carrier05.Lift_Info.TrayNot_Loaded_Lift2 := TRUE;
END_IF;
(* Rung 4: Settings Lift 04 *)
// Configuration settings
SettingsLift04.ActuatorBackOn:= TRUE;
SettingsLift04.ActuatorFrontOn:= TRUE;
SettingsLift04.ActuatorsLastPosition:= FALSE;
SettingsLift04.Option_InductiveTraydetection := TRUE;

// Instruction settings
IF (DatAControl_Lift04.IN.Instruction.Operand1 >= 1 OR DatAControl_Lift04.IN.Instruction.Operand1 <= 7) THEN
	SettingsLift04.PositionReferenceOk:= TRUE;
ELSE
	SettingsLift04.PositionReferenceOk:= FALSE;
END_IF;

IF DatAControl_Lift04.IN.Instruction.InstructionType= 4 AND (DatAControl_Lift04.IN.Instruction.Operand1 = 102 OR DatAControl_Lift04.IN.Instruction.Operand1 = 702) THEN
	SettingsLift04.UnloadGateOk:= TRUE;
ELSE
	SettingsLift04.UnloadGateOk:=FALSE;
END_IF;

IF DatAControl_Lift04.IN.Instruction.InstructionType= 3 AND (DatAControl_Lift04.IN.Instruction.Operand1 = 102 OR DatAControl_Lift04.IN.Instruction.Operand1 = 702) THEN
	SettingsLift04.LoadGateOk:= TRUE;
ELSE
	SettingsLift04.LoadGateOk:= FALSE;
END_IF;

// Parameters
SettingsLift04.MachineCode:=3;
SettingsLift04.SafeStopTime:=15;
SettingsLift04.Tolerance_At_Position:=25;
SettingsLift04.Warning_Tolerance_At_Position:=25;
SettingsLift04.BrakeReleaseFreq:=700;
SettingsLift04.Dec_Area_High:= 10000;
SettingsLift04.Dec_Area_Low:=1000;
SettingsLift04.NodeNummerLift:=9;
SettingsLift04.NodeNummerChain:=10;
SettingsLift04.MinimumSpeed:=1000;
SettingsLift04.MaximumSpeed:=8400; // Motor with extern brake 84Hz max, motor with no brake 87Hz max
SettingsLift04.MinimumSpeedChain:= 3700;
SettingsLift04.MaximumSpeedChain:= 8000; // Motor with intern brake 68 Hz max
SettingsLift04.TimeConFreeBackDOFF:= 50;
SettingsLift04.TimeConFreeBackDON:= 5;
SettingsLift04.TimeConFreeFrontDOFF:= 5;
SettingsLift04.TimeConFreeFrontDON:= 5;
SettingsLift04.UseBenchUnloadInstruction:= TRUE;

IF Commands_Lift04.Reverse THEN // Slow down
	SettingsLift04.MinimumSpeed := 750;
	SettingsLift04.BrakeReleaseFreq:=700;
END_IF;

IF SettingsLift04.Option_InductiveTraydetection THEN
	SettingsLift04.ChainHighSpeed := 60;
ELSE
 	SettingsLift04.ChainHighSpeed := 85;
END_IF;

SettingsLift04.TimeConInductiveBackDOFF := 2;
SettingsLift04.TimeConInductiveBackDON := 8;
SettingsLift04.TimeConInductiveFrontDOFF := 2;
SettingsLift04.TimeConInductiveFrontDON := 8;

// Mechanical settings
SettingsLift04.MinimumPulseLevel:=10000;
SettingsLift04.MaximumPulseLevel:=177000;
SettingsLift04.TooFarAllowed:= 1000;
SettingsLift04.ResetValueMargin := 500;
SettingsLift04.MinimumPosition:= 1;
SettingsLift04.MaximumPosition:= 10;
SettingsLift04.PulseLevel[1]:=10000;
SettingsLift04.PulseLevel[2]:= Lift4_PulsValueLevel2; // 13450;
SettingsLift04.PulseLevel[3]:= Lift4_PulsValueLevel3; // 25000;
SettingsLift04.PulseLevel[4]:= Lift4_PulsValueLevel4; // 53220;
SettingsLift04.PulseLevel[5]:= Lift4_PulsValueLevel5; // 73670;
SettingsLift04.PulseLevel[6]:= Lift4_PulsValueLevel6; // 94120;
SettingsLift04.PulseLevel[7]:= Lift4_PulsValueLevel7; // 114580;
SettingsLift04.PulseLevel[8]:= Lift4_PulsValueLevel8; // 135020;
SettingsLift04.PulseLevel[9]:= Lift4_PulsValueLevel9; // 155470;
SettingsLift04.PulseLevel[10]:= Lift4_PulsValueLevel10; // 175920;
SettingsLift04.PulseLevel[11]:=10;
SettingsLift04.PulseLevel[12]:=10;
SettingsLift04.PulseLevel[13]:=10;
SettingsLift04.PulseLevel[14]:=10;
SettingsLift04.PulseLevel[15]:=10;

SettingsLift04.NeedLevelSensor[1]:=TRUE;
SettingsLift04.NeedLevelSensor[2]:=FALSE;
SettingsLift04.NeedLevelSensor[3]:=FALSE;
SettingsLift04.NeedLevelSensor[4]:=TRUE;
SettingsLift04.NeedLevelSensor[5]:=TRUE;
SettingsLift04.NeedLevelSensor[6]:=TRUE;
SettingsLift04.NeedLevelSensor[7]:=TRUE;
SettingsLift04.NeedLevelSensor[8]:=TRUE;
SettingsLift04.NeedLevelSensor[9]:=TRUE;
SettingsLift04.NeedLevelSensor[10]:=TRUE;
SettingsLift04.NeedLevelSensor[11]:=TRUE;
SettingsLift04.NeedLevelSensor[12]:=TRUE;
SettingsLift04.NeedLevelSensor[13]:=TRUE;
SettingsLift04.NeedLevelSensor[14]:=TRUE;
SettingsLift04.NeedLevelSensor[15]:=TRUE;

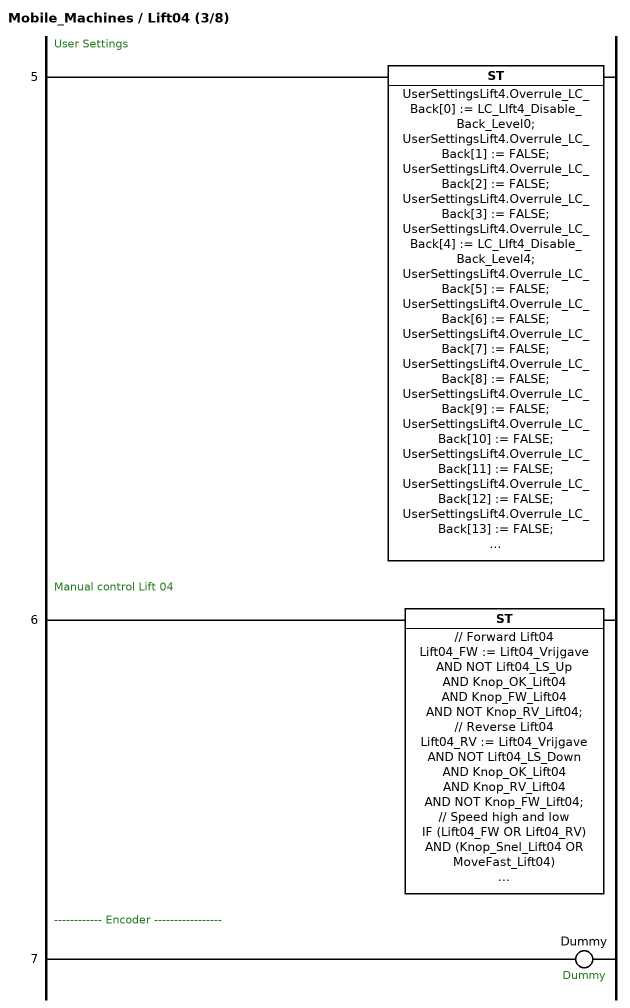
(* Rung 5: User Settings *)
UserSettingsLift4.Overrule_LC_Back[0] := LC_LIft4_Disable_Back_Level0;
UserSettingsLift4.Overrule_LC_Back[1] := FALSE;
UserSettingsLift4.Overrule_LC_Back[2] := FALSE;
UserSettingsLift4.Overrule_LC_Back[3] := FALSE;
UserSettingsLift4.Overrule_LC_Back[4] := LC_LIft4_Disable_Back_Level4;
UserSettingsLift4.Overrule_LC_Back[5] := FALSE;
UserSettingsLift4.Overrule_LC_Back[6] := FALSE;
UserSettingsLift4.Overrule_LC_Back[7] := FALSE;
UserSettingsLift4.Overrule_LC_Back[8] := FALSE;
UserSettingsLift4.Overrule_LC_Back[9] := FALSE;
UserSettingsLift4.Overrule_LC_Back[10] := FALSE;
UserSettingsLift4.Overrule_LC_Back[11] := FALSE;
UserSettingsLift4.Overrule_LC_Back[12] := FALSE;
UserSettingsLift4.Overrule_LC_Back[13] := FALSE;
UserSettingsLift4.Overrule_LC_Back[14] := FALSE;
UserSettingsLift4.Overrule_LC_Back[15] := FALSE;

UserSettingsLift4.Overrule_LC_Front[0] := LC_LIft4_Disable_Front_Level0;
UserSettingsLift4.Overrule_LC_Front[1] := LC_LIft4_Disable_Front_Level1;
UserSettingsLift4.Overrule_LC_Front[2] := LC_LIft4_Disable_Front_Level2;
UserSettingsLift4.Overrule_LC_Front[3] := LC_LIft4_Disable_Front_Level3;
UserSettingsLift4.Overrule_LC_Front[4] := LC_LIft4_Disable_Front_Level4;
UserSettingsLift4.Overrule_LC_Front[5] := LC_LIft4_Disable_Front_Level5;
UserSettingsLift4.Overrule_LC_Front[6] := LC_LIft4_Disable_Front_Level6;
UserSettingsLift4.Overrule_LC_Front[7] := LC_LIft4_Disable_Front_Level7;
UserSettingsLift4.Overrule_LC_Front[8] := FALSE;
UserSettingsLift4.Overrule_LC_Front[9] := FALSE;
UserSettingsLift4.Overrule_LC_Front[10] := FALSE;
UserSettingsLift4.Overrule_LC_Front[11] := FALSE;
UserSettingsLift4.Overrule_LC_Front[12] := FALSE;
UserSettingsLift4.Overrule_LC_Front[13] := FALSE;
UserSettingsLift4.Overrule_LC_Front[14] := FALSE;
UserSettingsLift4.Overrule_LC_Front[15] := FALSE;
(* Rung 6: Manual control Lift 04 *)
// Forward Lift04
Lift04_FW := Lift04_Vrijgave
AND NOT Lift04_LS_Up
AND Knop_OK_Lift04
AND Knop_FW_Lift04
AND NOT Knop_RV_Lift04;
// Reverse Lift04
Lift04_RV := Lift04_Vrijgave
AND NOT Lift04_LS_Down
AND Knop_OK_Lift04
AND Knop_RV_Lift04
AND NOT Knop_FW_Lift04;

// Speed high and low
IF (Lift04_FW OR Lift04_RV) AND (Knop_Snel_Lift04 OR MoveFast_Lift04)
AND EncoderLift04>SettingsLift04.MinimumPulseLevel+1000 AND EncoderLift04<SettingsLift04.MaximumPulseLevel-1000 THEN
	SettingsLift04.MinimumSpeed:=5000;
END_IF;

// Led ok Lift04
Led_Knop_OK_Lift04 := Knop_OK_Lift04 AND Lift04_Vrijgave;

// Vrijgave Lift04
Lift04_Vrijgave :=  (*Lift04_LS_FallProtect
AND*) Lift04_SafetyInput1 AND Lift04_SafetyInput2 AND Lift04_Alarms=0;

// Use manual control buttons as replacement for pocket (TEMP)
//Lift04_FW  Lift04_RV
IF Knop_OK_Lift04 THEN
	Pocket_Lift04.Move.Out:=Lift04_FW;
	Pocket_Lift04.Move.In:= Lift04_RV;
	Pocket_Lift04.Move.Stop:= NOT Lift04_FW AND NOT Lift04_RV;
END_IF;

// Move fast on/off
IF Pocket_Lift04.MoveFastOn THEN
	MoveFast_Lift04 := TRUE;
END_IF;
IF Pocket_Lift04.MoveFastOff OR DatAControl_Lift04.IN.MachineMode<>3 THEN
	MoveFast_Lift04 := FALSE;
END_IF;
Pocket_Lift04.MoveFastOn := FALSE;
Pocket_Lift04.MoveFastOff := FALSE;
(* Rung 7: ------------ Encoder ----------------- *)
Dummy := TRUE;

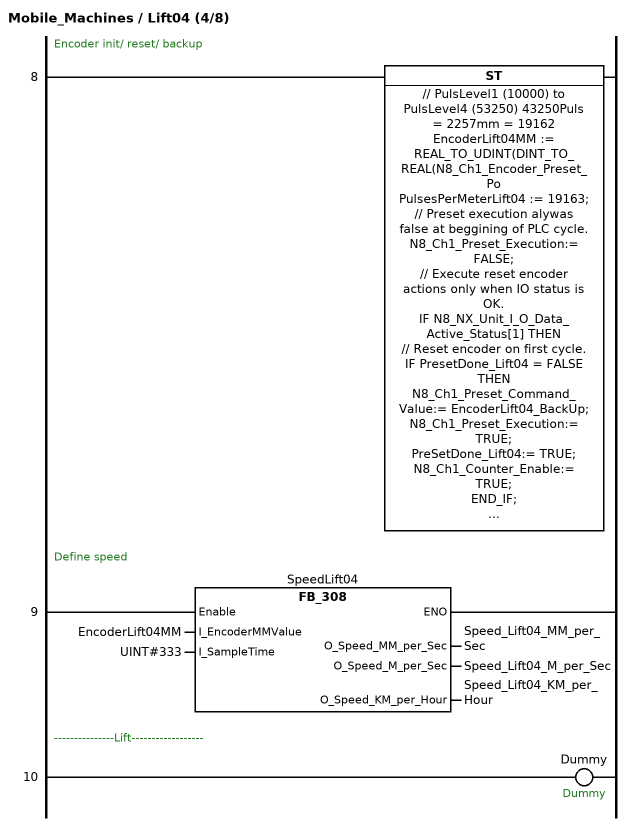
(* Rung 8: Encoder init/ reset/ backup *)
// PulsLevel1 (10000) to PulsLevel4 (53250) 43250Puls = 2257mm = 19162,605228179 PpM
EncoderLift04MM := REAL_TO_UDINT(DINT_TO_REAL(N8_Ch1_Encoder_Preset_Position) / UDINT_TO_REAL(PulsesPerMeterLift04) * 1000);
PulsesPerMeterLift04 := 19163;

// Preset execution alywas false at beggining of PLC cycle.
N8_Ch1_Preset_Execution:= FALSE;

// Execute reset encoder actions only when IO status is OK.
IF N8_NX_Unit_I_O_Data_Active_Status[1] THEN
	
	// Reset encoder on first cycle.
	IF PresetDone_Lift04 = FALSE THEN
		N8_Ch1_Preset_Command_Value:= EncoderLift04_BackUp;
		N8_Ch1_Preset_Execution:= TRUE;
		PreSetDone_Lift04:= TRUE;
		N8_Ch1_Counter_Enable:= TRUE;
	END_IF;
	
	// Reset encoder when lift is at position.
	IF ResetEncoder_Lift04  THEN
		N8_Ch1_Preset_Command_Value:= ResetEncoderValue_Lift04; // 10000 @Ground
		N8_Ch1_Preset_Execution:= TRUE;
		ResetEncoder_Lift04:= FALSE;
	END_IF;
	
	// Move encoder value.
    EncoderLift04 := DINT_TO_UDINT(N8_Ch1_Encoder_Preset_Position);
	
	// Backup encoder value.
	EncoderLift04_Backup:= EncoderLift04;
END_IF;
(* Rung 9: Define speed *)
SpeedLift04(Enable := TRUE, I_EncoderMMValue := EncoderLift04MM, I_SampleTime := UINT#333, O_Speed_MM_per_Sec => Speed_Lift04_MM_per_Sec, O_Speed_M_per_Sec => Speed_Lift04_M_per_Sec, O_Speed_KM_per_Hour => Speed_Lift04_KM_per_Hour);
(* Rung 10: ---------------Lift------------------ *)
Dummy := TRUE;

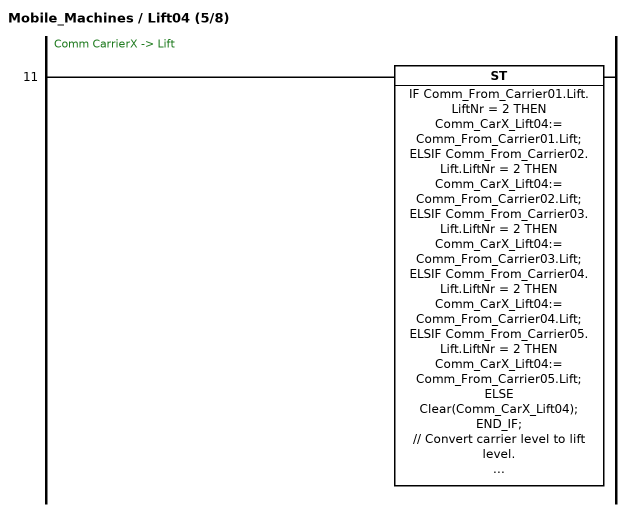
(* Rung 11: Comm CarrierX -> Lift *)
IF Comm_From_Carrier01.Lift.LiftNr = 2 THEN
	Comm_CarX_Lift04:= Comm_From_Carrier01.Lift;
ELSIF Comm_From_Carrier02.Lift.LiftNr = 2 THEN
	Comm_CarX_Lift04:= Comm_From_Carrier02.Lift;
ELSIF Comm_From_Carrier03.Lift.LiftNr = 2 THEN
	Comm_CarX_Lift04:= Comm_From_Carrier03.Lift;
ELSIF Comm_From_Carrier04.Lift.LiftNr = 2 THEN
	Comm_CarX_Lift04:= Comm_From_Carrier04.Lift;
ELSIF Comm_From_Carrier05.Lift.LiftNr = 2 THEN
	Comm_CarX_Lift04:= Comm_From_Carrier05.Lift;
ELSE
	Clear(Comm_CarX_Lift04);
END_IF;

// Convert carrier level to lift level.
//This is only needed when lift has more levels than the carrier!
CASE Comm_CarX_Lift04.Height_MobileMachine OF
	1: Comm_CarX_Lift04.Height_MobileMachine:=4;
	2: Comm_CarX_Lift04.Height_MobileMachine:=5;
	// mezzanine will probably add an extra level to the lift ones.
	3: Comm_CarX_Lift04.Height_MobileMachine:=6;
	4: Comm_CarX_Lift04.Height_MobileMachine:=7;
	5: Comm_CarX_Lift04.Height_MobileMachine:=8;
	6: Comm_CarX_Lift04.Height_MobileMachine:=9;
	7: Comm_CarX_Lift04.Height_MobileMachine:=10;
ELSE
	// If lift drops the carrier on a level not listed above set to 0 to avoid wrong positions.
     Comm_CarX_Lift04.Height_MobileMachine:=0;
END_CASE;

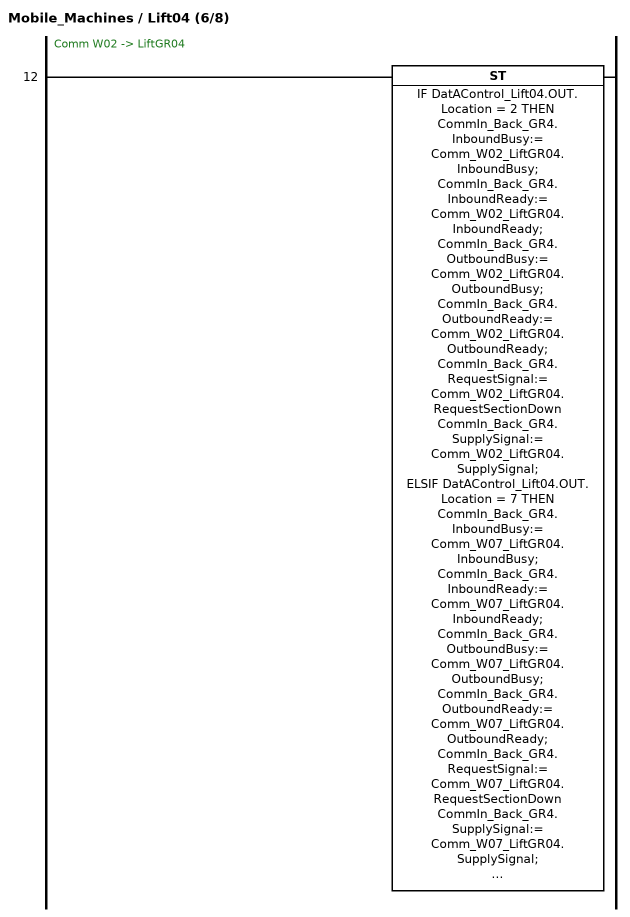
(* Rung 12: Comm W02 -> LiftGR04 *)
IF DatAControl_Lift04.OUT.Location = 2 THEN
	CommIn_Back_GR4.InboundBusy:= Comm_W02_LiftGR04.InboundBusy;
	CommIn_Back_GR4.InboundReady:= Comm_W02_LiftGR04.InboundReady;
	CommIn_Back_GR4.OutboundBusy:= Comm_W02_LiftGR04.OutboundBusy;
	CommIn_Back_GR4.OutboundReady:= Comm_W02_LiftGR04.OutboundReady;
	CommIn_Back_GR4.RequestSignal:= Comm_W02_LiftGR04.RequestSectionDown;
	CommIn_Back_GR4.SupplySignal:= Comm_W02_LiftGR04.SupplySignal;
ELSIF DatAControl_Lift04.OUT.Location = 7 THEN
	CommIn_Back_GR4.InboundBusy:= Comm_W07_LiftGR04.InboundBusy;
	CommIn_Back_GR4.InboundReady:= Comm_W07_LiftGR04.InboundReady;
	CommIn_Back_GR4.OutboundBusy:= Comm_W07_LiftGR04.OutboundBusy;
	CommIn_Back_GR4.OutboundReady:= Comm_W07_LiftGR04.OutboundReady;
	CommIn_Back_GR4.RequestSignal:= Comm_W07_LiftGR04.RequestSectionDown;
	CommIn_Back_GR4.SupplySignal:= Comm_W07_LiftGR04.SupplySignal;
END_IF;

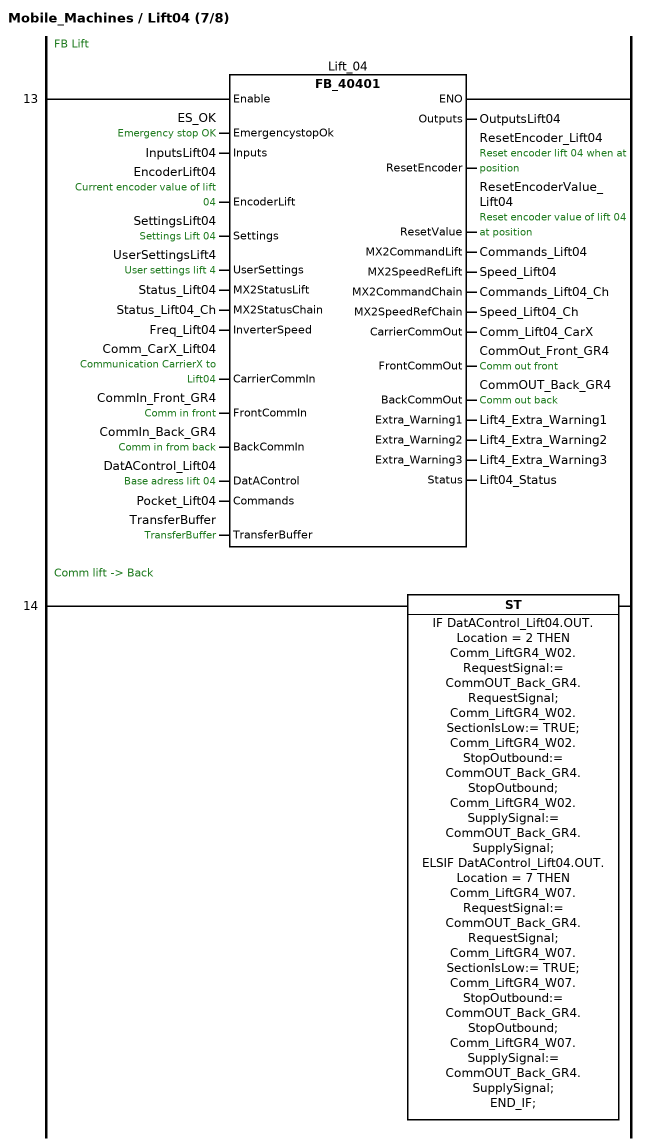
(* Rung 13: FB Lift *)
Lift_04(Enable := TRUE, EmergencystopOk := ES_OK, Inputs := InputsLift04, EncoderLift := EncoderLift04, Settings := SettingsLift04, UserSettings := UserSettingsLift4, MX2StatusLift := Status_Lift04, MX2StatusChain := Status_Lift04_Ch, InverterSpeed := Freq_Lift04, CarrierCommIn := Comm_CarX_Lift04, FrontCommIn := CommIn_Front_GR4, BackCommIn := CommIn_Back_GR4, DatAControl := DatAControl_Lift04, Commands := Pocket_Lift04, TransferBuffer := TransferBuffer, Outputs => OutputsLift04, ResetEncoder => ResetEncoder_Lift04, ResetValue => ResetEncoderValue_Lift04, MX2CommandLift => Commands_Lift04, MX2SpeedRefLift => Speed_Lift04, MX2CommandChain => Commands_Lift04_Ch, MX2SpeedRefChain => Speed_Lift04_Ch, CarrierCommOut => Comm_Lift04_CarX, FrontCommOut => CommOut_Front_GR4, BackCommOut => CommOUT_Back_GR4, Extra_Warning1 => Lift4_Extra_Warning1, Extra_Warning2 => Lift4_Extra_Warning2, Extra_Warning3 => Lift4_Extra_Warning3, Status => Lift04_Status);
(* Rung 14: Comm lift -> Back *)
IF DatAControl_Lift04.OUT.Location = 2 THEN
Comm_LiftGR4_W02.RequestSignal:= CommOUT_Back_GR4.RequestSignal;
Comm_LiftGR4_W02.SectionIsLow:= TRUE;
Comm_LiftGR4_W02.StopOutbound:= CommOUT_Back_GR4.StopOutbound;
Comm_LiftGR4_W02.SupplySignal:= CommOUT_Back_GR4.SupplySignal;
ELSIF DatAControl_Lift04.OUT.Location = 7 THEN
Comm_LiftGR4_W07.RequestSignal:= CommOUT_Back_GR4.RequestSignal;
Comm_LiftGR4_W07.SectionIsLow:= TRUE;
Comm_LiftGR4_W07.StopOutbound:= CommOUT_Back_GR4.StopOutbound;
Comm_LiftGR4_W07.SupplySignal:= CommOUT_Back_GR4.SupplySignal;
END_IF;

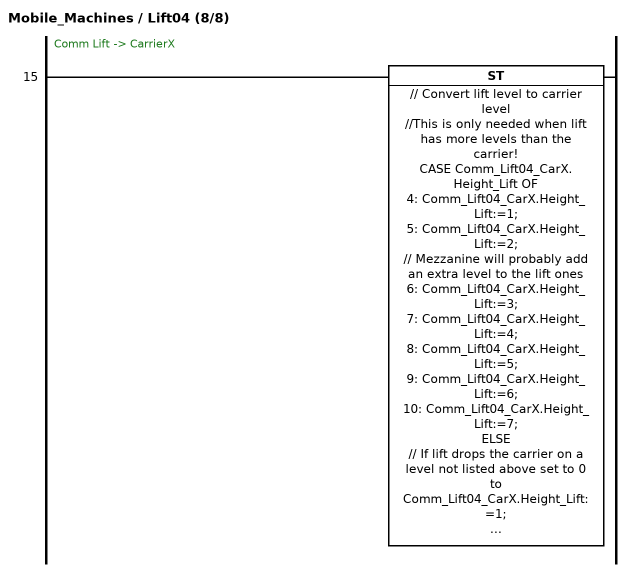
(* Rung 15: Comm Lift -> CarrierX *)
// Convert lift level to carrier level
//This is only needed when lift has more levels than the carrier!
CASE Comm_Lift04_CarX.Height_Lift OF
	4: Comm_Lift04_CarX.Height_Lift:=1;
	5: Comm_Lift04_CarX.Height_Lift:=2;
	// Mezzanine will probably add an extra level to the lift ones
	6: Comm_Lift04_CarX.Height_Lift:=3;
	7: Comm_Lift04_CarX.Height_Lift:=4;
	8: Comm_Lift04_CarX.Height_Lift:=5;
	9: Comm_Lift04_CarX.Height_Lift:=6;
	10: Comm_Lift04_CarX.Height_Lift:=7;
ELSE
	// If lift drops the carrier on a level not listed above set to 0 to avoid wrong positions.
     Comm_Lift04_CarX.Height_Lift:=1;
END_CASE;

IF Comm_From_Carrier01.Lift.LiftNr = 2 THEN
	Comm_To_Carrier01.Lift:= Comm_Lift04_CarX;
ELSIF Comm_From_Carrier02.Lift.LiftNr = 2 THEN
	Comm_To_Carrier02.Lift:= Comm_Lift04_CarX;
ELSIF Comm_From_Carrier03.Lift.LiftNr = 2 THEN
	Comm_To_Carrier03.Lift:= Comm_Lift04_CarX;
ELSIF Comm_From_Carrier04.Lift.LiftNr = 2 THEN
	Comm_To_Carrier04.Lift:= Comm_Lift04_CarX;
ELSIF Comm_From_Carrier05.Lift.LiftNr = 2 THEN
	Comm_To_Carrier05.Lift:= Comm_Lift04_CarX;
END_IF;

(* Section Carrier01: ladder, written here as Structured Text *)

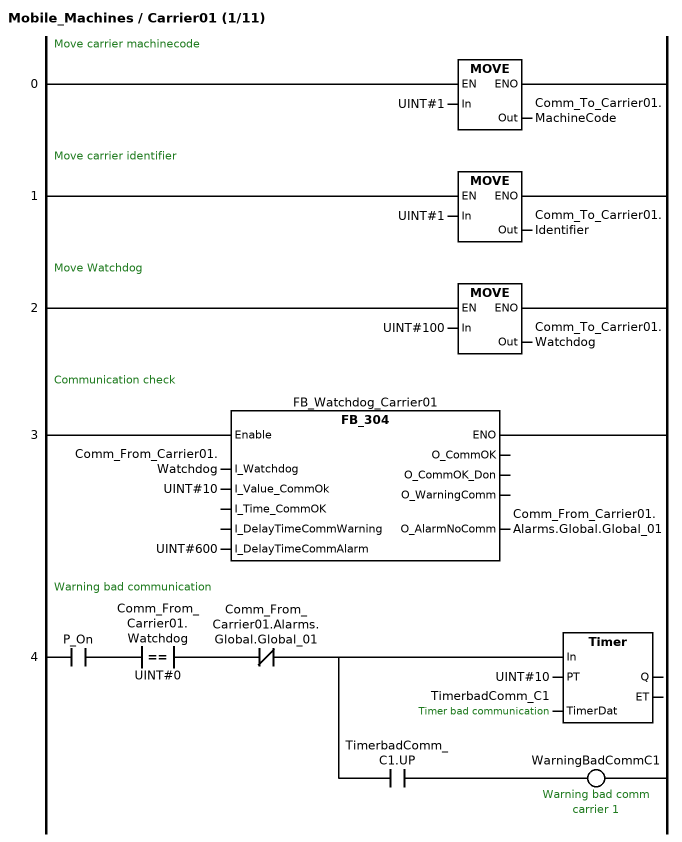
(* Rung 0: Move carrier machinecode *)
Comm_To_Carrier01.MachineCode := UINT#1;
(* Rung 1: Move carrier identifier *)
Comm_To_Carrier01.Identifier := UINT#1;
(* Rung 2: Move Watchdog *)
Comm_To_Carrier01.Watchdog := UINT#100;
(* Rung 3: Communication check *)
FB_Watchdog_Carrier01(Enable := TRUE, I_Watchdog := Comm_From_Carrier01.Watchdog, I_Value_CommOk := UINT#10, I_DelayTimeCommAlarm := UINT#600, O_AlarmNoComm => Comm_From_Carrier01.Alarms.Global.Global_01);
(* Rung 4: Warning bad communication *)
_p1 := P_On AND (Comm_From_Carrier01.Watchdog = UINT#0) AND NOT Comm_From_Carrier01.Alarms.Global.Global_01;
_t2 := Timer(In := _p1, PT := UINT#10, TimerDat := TimerbadComm_C1);
WarningBadCommC1 := _p1 AND TimerbadComm_C1.UP;

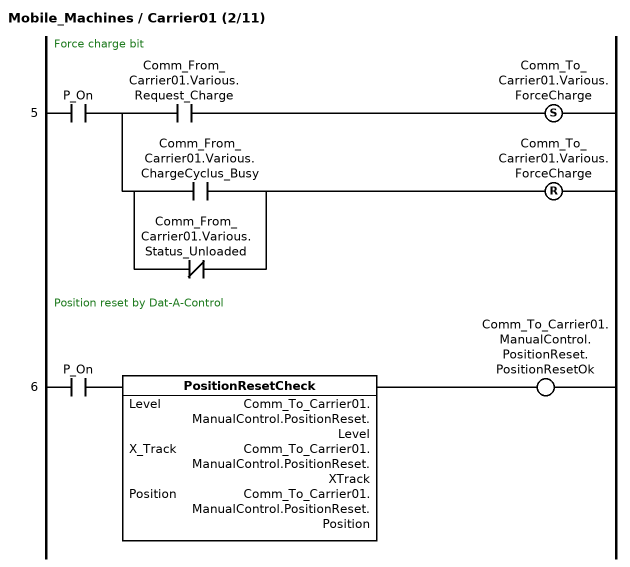
(* Rung 5: Force charge bit *)
IF P_On AND Comm_From_Carrier01.Various.Request_Charge THEN
    Comm_To_Carrier01.Various.ForceCharge := TRUE;
END_IF;
IF P_On AND (Comm_From_Carrier01.Various.ChargeCyclus_Busy OR NOT Comm_From_Carrier01.Various.Status_Unloaded) THEN
    Comm_To_Carrier01.Various.ForceCharge := FALSE;
END_IF;
(* Rung 6: Position reset by Dat-A-Control *)
Comm_To_Carrier01.ManualControl.PositionReset.PositionResetOk := P_On AND PositionResetCheck(Level := Comm_To_Carrier01.ManualControl.PositionReset.Level, X_Track := Comm_To_Carrier01.ManualControl.PositionReset.XTrack, Position := Comm_To_Carrier01.ManualControl.PositionReset.Position);

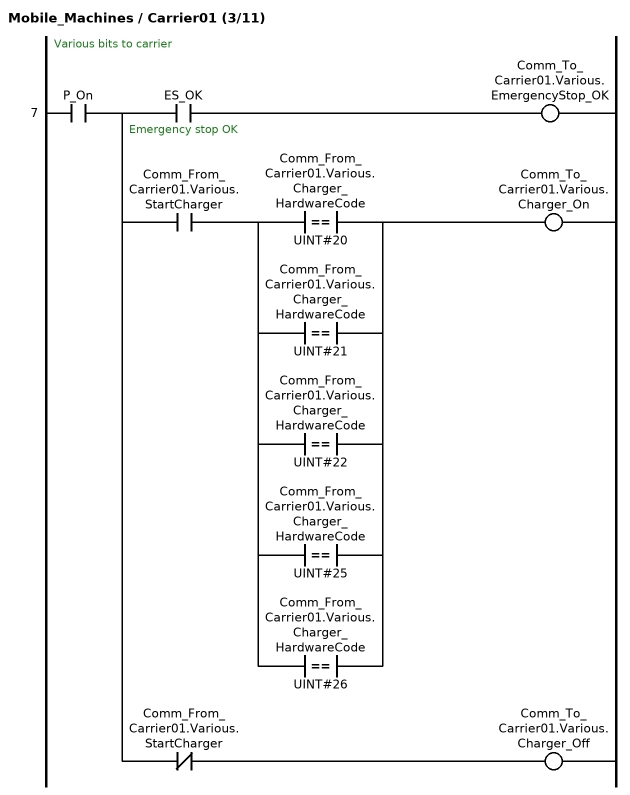
(* Rung 7: Various bits to carrier *)
Comm_To_Carrier01.Various.EmergencyStop_OK := P_On AND ES_OK;
Comm_To_Carrier01.Various.Charger_On := P_On AND Comm_From_Carrier01.Various.StartCharger AND ((Comm_From_Carrier01.Various.Charger_HardwareCode = UINT#20) OR (Comm_From_Carrier01.Various.Charger_HardwareCode = UINT#21) OR (Comm_From_Carrier01.Various.Charger_HardwareCode = UINT#22) OR (Comm_From_Carrier01.Various.Charger_HardwareCode = UINT#25) OR (Comm_From_Carrier01.Various.Charger_HardwareCode = UINT#26));
Comm_To_Carrier01.Various.Charger_Off := P_On AND NOT Comm_From_Carrier01.Various.StartCharger;

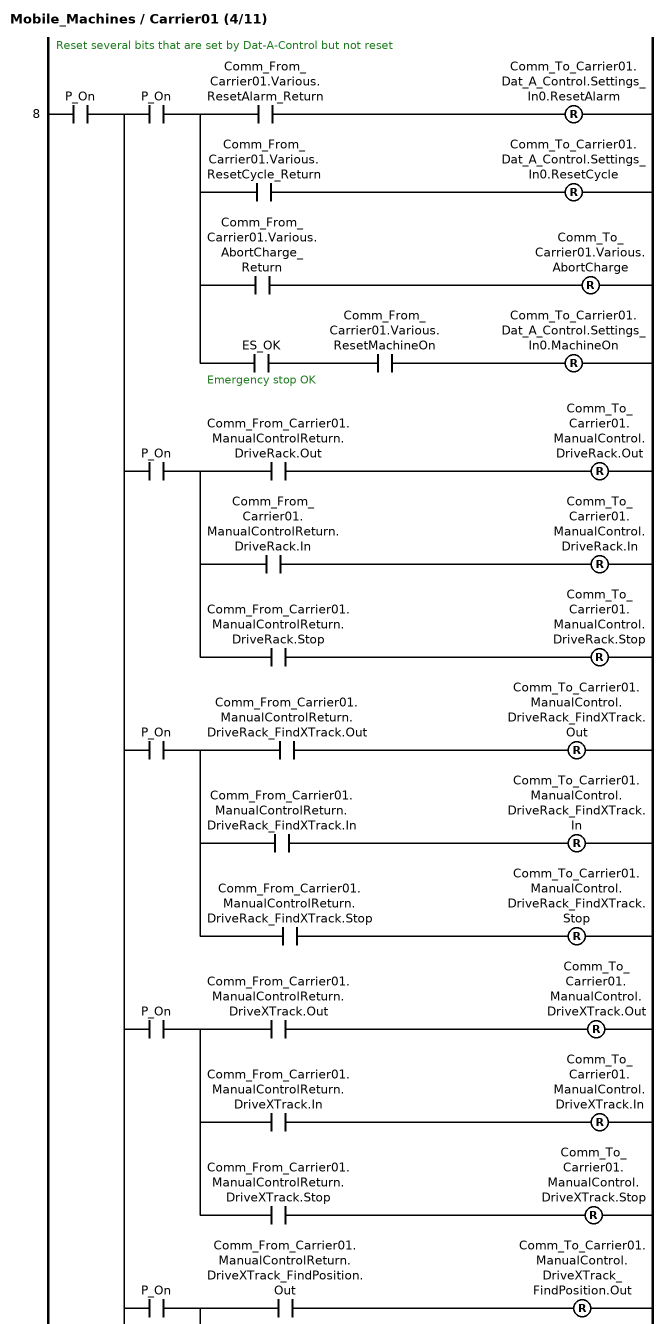

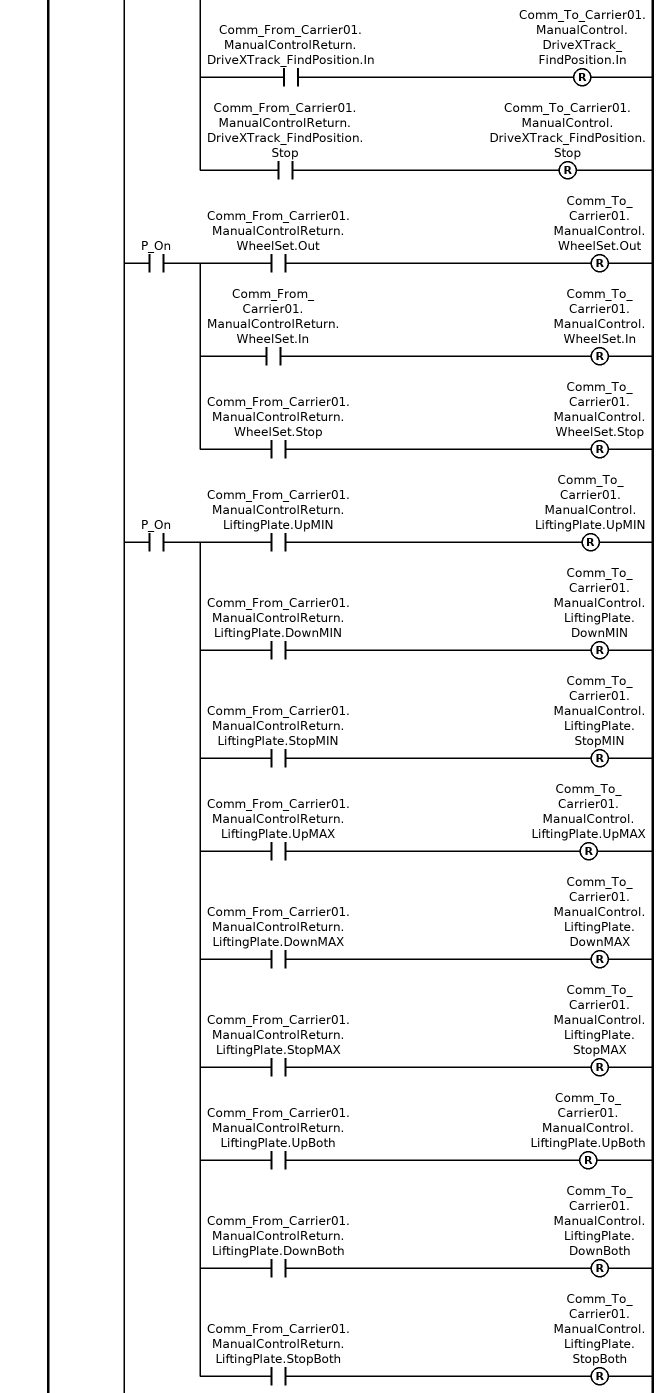

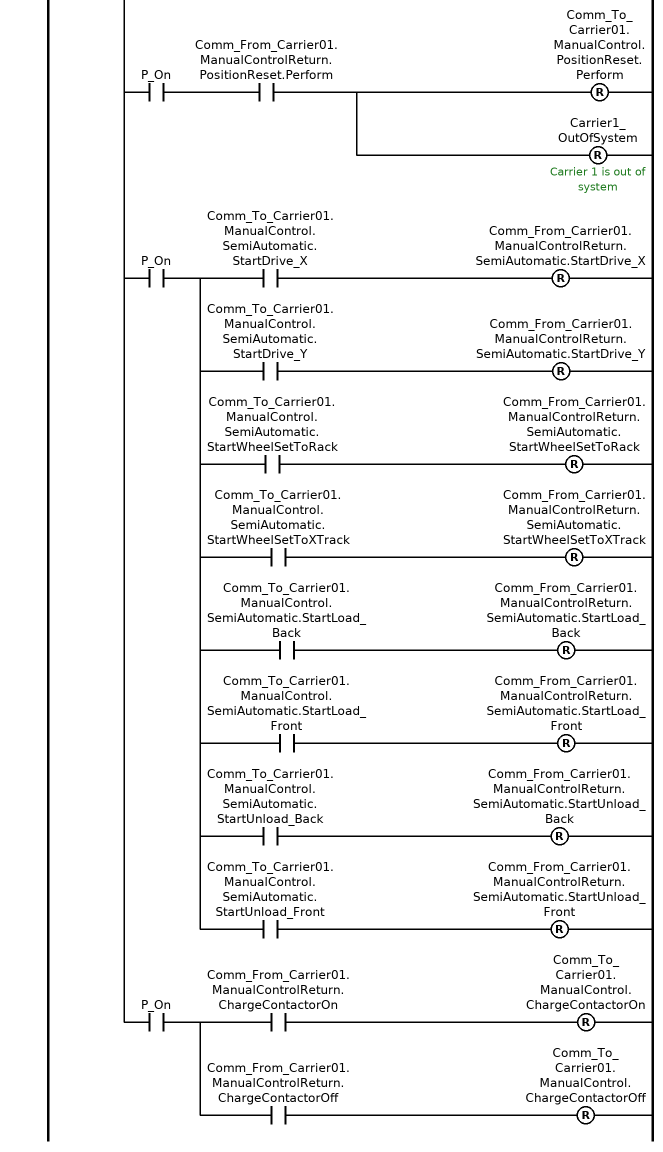
(* Rung 8: Reset several bits that are set by Dat-A-Control but not reset *)
IF P_On AND P_On AND Comm_From_Carrier01.Various.ResetAlarm_Return THEN
    Comm_To_Carrier01.Dat_A_Control.Settings_In0.ResetAlarm := FALSE;
END_IF;
IF P_On AND P_On AND Comm_From_Carrier01.Various.ResetCycle_Return THEN
    Comm_To_Carrier01.Dat_A_Control.Settings_In0.ResetCycle := FALSE;
END_IF;
IF P_On AND P_On AND Comm_From_Carrier01.Various.AbortCharge_Return THEN
    Comm_To_Carrier01.Various.AbortCharge := FALSE;
END_IF;
IF P_On AND P_On AND ES_OK AND Comm_From_Carrier01.Various.ResetMachineOn THEN
    Comm_To_Carrier01.Dat_A_Control.Settings_In0.MachineOn := FALSE;
END_IF;
IF P_On AND P_On AND Comm_From_Carrier01.ManualControlReturn.DriveRack.Out THEN
    Comm_To_Carrier01.ManualControl.DriveRack.Out := FALSE;
END_IF;
IF P_On AND P_On AND Comm_From_Carrier01.ManualControlReturn.DriveRack.In THEN
    Comm_To_Carrier01.ManualControl.DriveRack.In := FALSE;
END_IF;
IF P_On AND P_On AND Comm_From_Carrier01.ManualControlReturn.DriveRack.Stop THEN
    Comm_To_Carrier01.ManualControl.DriveRack.Stop := FALSE;
END_IF;
IF P_On AND P_On AND Comm_From_Carrier01.ManualControlReturn.DriveRack_FindXTrack.Out THEN
    Comm_To_Carrier01.ManualControl.DriveRack_FindXTrack.Out := FALSE;
END_IF;
IF P_On AND P_On AND Comm_From_Carrier01.ManualControlReturn.DriveRack_FindXTrack.In THEN
    Comm_To_Carrier01.ManualControl.DriveRack_FindXTrack.In := FALSE;
END_IF;
IF P_On AND P_On AND Comm_From_Carrier01.ManualControlReturn.DriveRack_FindXTrack.Stop THEN
    Comm_To_Carrier01.ManualControl.DriveRack_FindXTrack.Stop := FALSE;
END_IF;
IF P_On AND P_On AND Comm_From_Carrier01.ManualControlReturn.DriveXTrack.Out THEN
    Comm_To_Carrier01.ManualControl.DriveXTrack.Out := FALSE;
END_IF;
IF P_On AND P_On AND Comm_From_Carrier01.ManualControlReturn.DriveXTrack.In THEN
    Comm_To_Carrier01.ManualControl.DriveXTrack.In := FALSE;
END_IF;
IF P_On AND P_On AND Comm_From_Carrier01.ManualControlReturn.DriveXTrack.Stop THEN
    Comm_To_Carrier01.ManualControl.DriveXTrack.Stop := FALSE;
END_IF;
IF P_On AND P_On AND Comm_From_Carrier01.ManualControlReturn.DriveXTrack_FindPosition.Out THEN
    Comm_To_Carrier01.ManualControl.DriveXTrack_FindPosition.Out := FALSE;
END_IF;
IF P_On AND P_On AND Comm_From_Carrier01.ManualControlReturn.DriveXTrack_FindPosition.In THEN
    Comm_To_Carrier01.ManualControl.DriveXTrack_FindPosition.In := FALSE;
END_IF;
IF P_On AND P_On AND Comm_From_Carrier01.ManualControlReturn.DriveXTrack_FindPosition.Stop THEN
    Comm_To_Carrier01.ManualControl.DriveXTrack_FindPosition.Stop := FALSE;
END_IF;
IF P_On AND P_On AND Comm_From_Carrier01.ManualControlReturn.WheelSet.Out THEN
    Comm_To_Carrier01.ManualControl.WheelSet.Out := FALSE;
END_IF;
IF P_On AND P_On AND Comm_From_Carrier01.ManualControlReturn.WheelSet.In THEN
    Comm_To_Carrier01.ManualControl.WheelSet.In := FALSE;
END_IF;
IF P_On AND P_On AND Comm_From_Carrier01.ManualControlReturn.WheelSet.Stop THEN
    Comm_To_Carrier01.ManualControl.WheelSet.Stop := FALSE;
END_IF;
IF P_On AND P_On AND Comm_From_Carrier01.ManualControlReturn.LiftingPlate.UpMIN THEN
    Comm_To_Carrier01.ManualControl.LiftingPlate.UpMIN := FALSE;
END_IF;
IF P_On AND P_On AND Comm_From_Carrier01.ManualControlReturn.LiftingPlate.DownMIN THEN
    Comm_To_Carrier01.ManualControl.LiftingPlate.DownMIN := FALSE;
END_IF;
IF P_On AND P_On AND Comm_From_Carrier01.ManualControlReturn.LiftingPlate.StopMIN THEN
    Comm_To_Carrier01.ManualControl.LiftingPlate.StopMIN := FALSE;
END_IF;
IF P_On AND P_On AND Comm_From_Carrier01.ManualControlReturn.LiftingPlate.UpMAX THEN
    Comm_To_Carrier01.ManualControl.LiftingPlate.UpMAX := FALSE;
END_IF;
IF P_On AND P_On AND Comm_From_Carrier01.ManualControlReturn.LiftingPlate.DownMAX THEN
    Comm_To_Carrier01.ManualControl.LiftingPlate.DownMAX := FALSE;
END_IF;
IF P_On AND P_On AND Comm_From_Carrier01.ManualControlReturn.LiftingPlate.StopMAX THEN
    Comm_To_Carrier01.ManualControl.LiftingPlate.StopMAX := FALSE;
END_IF;
IF P_On AND P_On AND Comm_From_Carrier01.ManualControlReturn.LiftingPlate.UpBoth THEN
    Comm_To_Carrier01.ManualControl.LiftingPlate.UpBoth := FALSE;
END_IF;
IF P_On AND P_On AND Comm_From_Carrier01.ManualControlReturn.LiftingPlate.DownBoth THEN
    Comm_To_Carrier01.ManualControl.LiftingPlate.DownBoth := FALSE;
END_IF;
IF P_On AND P_On AND Comm_From_Carrier01.ManualControlReturn.LiftingPlate.StopBoth THEN
    Comm_To_Carrier01.ManualControl.LiftingPlate.StopBoth := FALSE;
END_IF;
_p3 := P_On AND P_On AND Comm_From_Carrier01.ManualControlReturn.PositionReset.Perform;
IF _p3 THEN
    Comm_To_Carrier01.ManualControl.PositionReset.Perform := FALSE;
    Carrier1_OutOfSystem := FALSE;
END_IF;
IF P_On AND P_On AND Comm_To_Carrier01.ManualControl.SemiAutomatic.StartDrive_X THEN
    Comm_From_Carrier01.ManualControlReturn.SemiAutomatic.StartDrive_X := FALSE;
END_IF;
IF P_On AND P_On AND Comm_To_Carrier01.ManualControl.SemiAutomatic.StartDrive_Y THEN
    Comm_From_Carrier01.ManualControlReturn.SemiAutomatic.StartDrive_Y := FALSE;
END_IF;
IF P_On AND P_On AND Comm_To_Carrier01.ManualControl.SemiAutomatic.StartWheelSetToRack THEN
    Comm_From_Carrier01.ManualControlReturn.SemiAutomatic.StartWheelSetToRack := FALSE;
END_IF;
IF P_On AND P_On AND Comm_To_Carrier01.ManualControl.SemiAutomatic.StartWheelSetToXTrack THEN
    Comm_From_Carrier01.ManualControlReturn.SemiAutomatic.StartWheelSetToXTrack := FALSE;
END_IF;
IF P_On AND P_On AND Comm_To_Carrier01.ManualControl.SemiAutomatic.StartLoad_Back THEN
    Comm_From_Carrier01.ManualControlReturn.SemiAutomatic.StartLoad_Back := FALSE;
END_IF;
IF P_On AND P_On AND Comm_To_Carrier01.ManualControl.SemiAutomatic.StartLoad_Front THEN
    Comm_From_Carrier01.ManualControlReturn.SemiAutomatic.StartLoad_Front := FALSE;
END_IF;
IF P_On AND P_On AND Comm_To_Carrier01.ManualControl.SemiAutomatic.StartUnload_Back THEN
    Comm_From_Carrier01.ManualControlReturn.SemiAutomatic.StartUnload_Back := FALSE;
END_IF;
IF P_On AND P_On AND Comm_To_Carrier01.ManualControl.SemiAutomatic.StartUnload_Front THEN
    Comm_From_Carrier01.ManualControlReturn.SemiAutomatic.StartUnload_Front := FALSE;
END_IF;
IF P_On AND P_On AND Comm_From_Carrier01.ManualControlReturn.ChargeContactorOn THEN
    Comm_To_Carrier01.ManualControl.ChargeContactorOn := FALSE;
END_IF;
IF P_On AND P_On AND Comm_From_Carrier01.ManualControlReturn.ChargeContactorOff THEN
    Comm_To_Carrier01.ManualControl.ChargeContactorOff := FALSE;
END_IF;

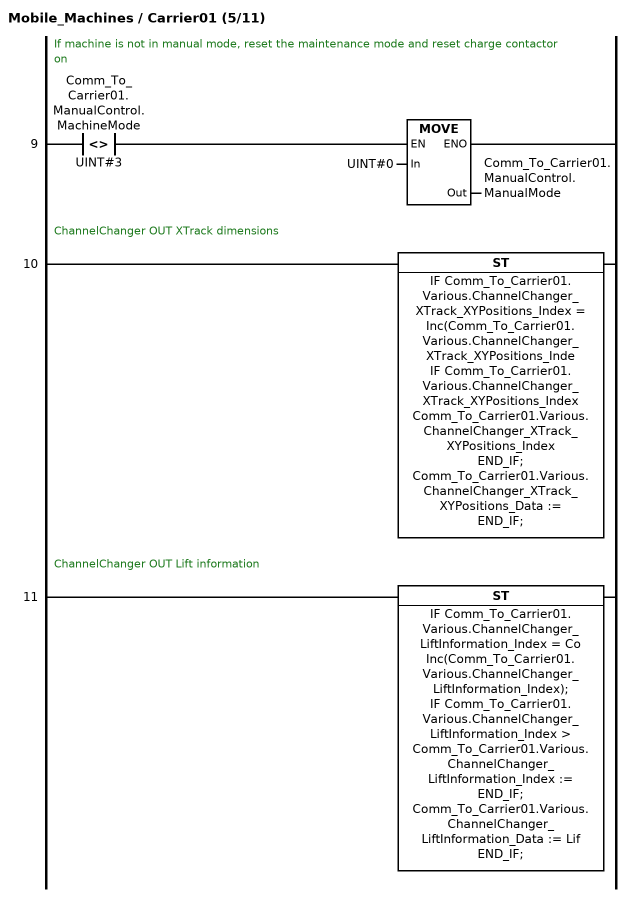
(* Rung 9: If machine is not in manual mode, reset the maintenance mode and reset charge contactor on *)
IF Comm_To_Carrier01.ManualControl.MachineMode <> UINT#3 THEN
    Comm_To_Carrier01.ManualControl.ManualMode := UINT#0;
END_IF;
(* Rung 10: ChannelChanger OUT XTrack dimensions *)
IF Comm_To_Carrier01.Various.ChannelChanger_XTrack_XYPositions_Index = Comm_From_Carrier01.Various.ChannelChanger_XTrack_XYPositions_Index THEN
	Inc(Comm_To_Carrier01.Various.ChannelChanger_XTrack_XYPositions_Index);
	IF Comm_To_Carrier01.Various.ChannelChanger_XTrack_XYPositions_Index > 199 THEN
		Comm_To_Carrier01.Various.ChannelChanger_XTrack_XYPositions_Index := 0;
	END_IF;
	Comm_To_Carrier01.Various.ChannelChanger_XTrack_XYPositions_Data := XTrack_XYPositions_Array[Comm_To_Carrier01.Various.ChannelChanger_XTrack_XYPositions_Index];
END_IF;
(* Rung 11: ChannelChanger OUT Lift information *)
IF Comm_To_Carrier01.Various.ChannelChanger_LiftInformation_Index = Comm_From_Carrier01.Various.ChannelChanger_LiftInformation_Index THEN
	Inc(Comm_To_Carrier01.Various.ChannelChanger_LiftInformation_Index);
	IF Comm_To_Carrier01.Various.ChannelChanger_LiftInformation_Index > 99 THEN
		Comm_To_Carrier01.Various.ChannelChanger_LiftInformation_Index := 0;
	END_IF;
	Comm_To_Carrier01.Various.ChannelChanger_LiftInformation_Data := Lift_Array[Comm_To_Carrier01.Various.ChannelChanger_LiftInformation_Index];
END_IF;

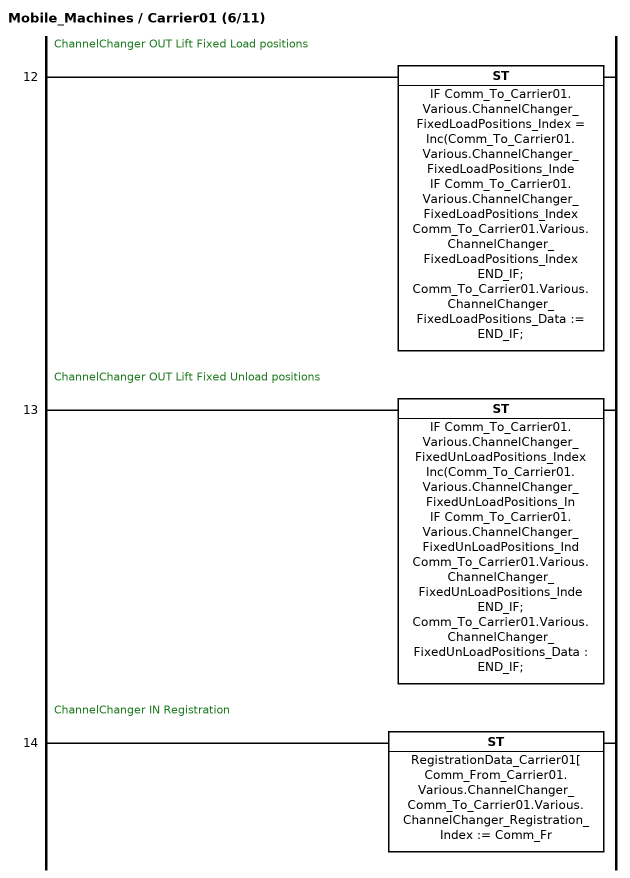
(* Rung 12: ChannelChanger OUT Lift Fixed Load positions *)
IF Comm_To_Carrier01.Various.ChannelChanger_FixedLoadPositions_Index = Comm_From_Carrier01.Various.ChannelChanger_FixedLoadPositions_Index THEN
	Inc(Comm_To_Carrier01.Various.ChannelChanger_FixedLoadPositions_Index);
	IF Comm_To_Carrier01.Various.ChannelChanger_FixedLoadPositions_Index > 199 THEN
		Comm_To_Carrier01.Various.ChannelChanger_FixedLoadPositions_Index := 0;
	END_IF;
	Comm_To_Carrier01.Various.ChannelChanger_FixedLoadPositions_Data := FixedLoadPosition_Array[Comm_To_Carrier01.Various.ChannelChanger_FixedLoadPositions_Index];
END_IF;
(* Rung 13: ChannelChanger OUT Lift Fixed Unload positions *)
IF Comm_To_Carrier01.Various.ChannelChanger_FixedUnLoadPositions_Index = Comm_From_Carrier01.Various.ChannelChanger_FixedUnLoadPositions_Index THEN
	Inc(Comm_To_Carrier01.Various.ChannelChanger_FixedUnLoadPositions_Index);
	IF Comm_To_Carrier01.Various.ChannelChanger_FixedUnLoadPositions_Index > 199 THEN
		Comm_To_Carrier01.Various.ChannelChanger_FixedUnLoadPositions_Index := 0;
	END_IF;
	Comm_To_Carrier01.Various.ChannelChanger_FixedUnLoadPositions_Data := FixedUnloadPosition_Array[Comm_To_Carrier01.Various.ChannelChanger_FixedUnLoadPositions_Index];
END_IF;
(* Rung 14: ChannelChanger IN Registration *)
RegistrationData_Carrier01[Comm_From_Carrier01.Various.ChannelChanger_Registration_Index] := Comm_From_Carrier01.Various.ChannelChanger_Registration_Data;
Comm_To_Carrier01.Various.ChannelChanger_Registration_Index := Comm_From_Carrier01.Various.ChannelChanger_Registration_Index;

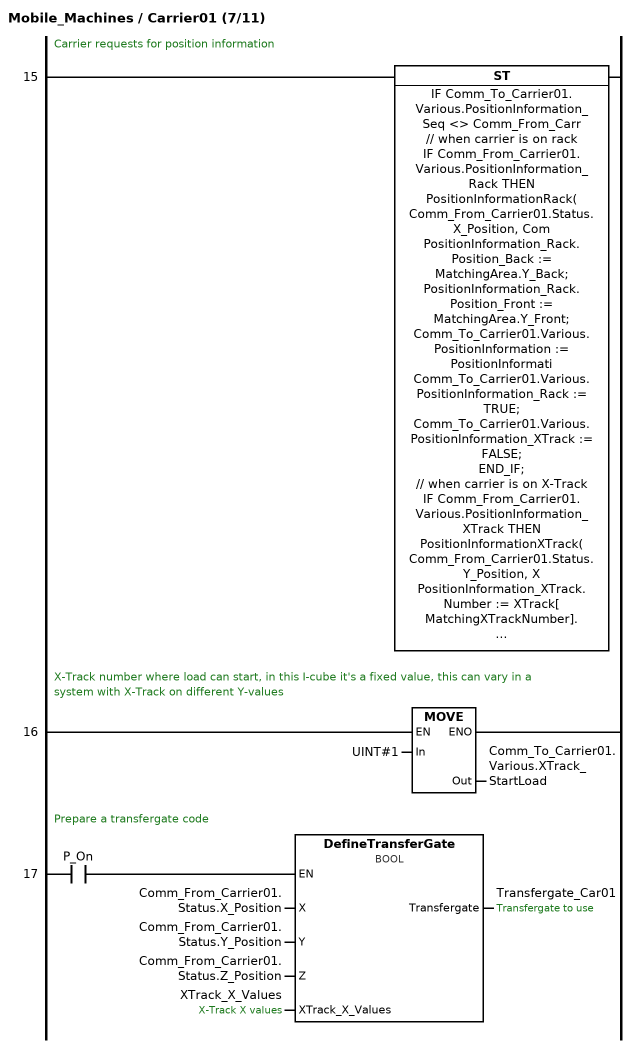
(* Rung 15: Carrier requests for position information *)
IF Comm_To_Carrier01.Various.PositionInformation_Seq <> Comm_From_Carrier01.Various.PositionInformation_Seq THEN
	// when carrier is on rack
	IF Comm_From_Carrier01.Various.PositionInformation_Rack THEN
		PositionInformationRack(Comm_From_Carrier01.Status.X_Position, Comm_From_Carrier01.Status.Y_Position, Comm_From_Carrier01.Status.Z_Position, Settings_CP.Margin_AreaCompare, Area, MatchingArea);
		PositionInformation_Rack.Position_Back := MatchingArea.Y_Back;
		PositionInformation_Rack.Position_Front := MatchingArea.Y_Front;
		Comm_To_Carrier01.Various.PositionInformation := PositionInformation_Rough;
		Comm_To_Carrier01.Various.PositionInformation_Rack := TRUE;
		Comm_To_Carrier01.Various.PositionInformation_XTrack := FALSE;
	END_IF;
	
	// when carrier is on X-Track
	IF Comm_From_Carrier01.Various.PositionInformation_XTrack THEN
		PositionInformationXTrack(Comm_From_Carrier01.Status.Y_Position, XTrack_Y_Values, MatchingXTrackNumber);
		PositionInformation_XTrack.Number := XTrack[MatchingXTrackNumber].XTrack_Number;
		PositionInformation_XTrack.Position_MIN := XTrack[MatchingXTrackNumber].MinimumPosition;
		PositionInformation_XTrack.Position_MAX := XTrack[MatchingXTrackNumber].MaximumPosition;
		Comm_To_Carrier01.Various.PositionInformation := PositionInformation_Rough;
		Comm_To_Carrier01.Various.PositionInformation_Rack := FALSE;
		Comm_To_Carrier01.Various.PositionInformation_XTrack := TRUE;
	END_IF;
	
	Comm_To_Carrier01.Various.PositionInformation_Seq := Comm_From_Carrier01.Various.PositionInformation_Seq;
	
END_IF;
(* Rung 16: X-Track number where load can start, in this I-cube it's a fixed value, this can vary in a system with X-Track on different Y-values *)
Comm_To_Carrier01.Various.XTrack_StartLoad := UINT#1;
(* Rung 17: Prepare a transfergate code *)
_t4 := FALSE;
IF P_On THEN _t4 := DefineTransferGate(X := Comm_From_Carrier01.Status.X_Position, Y := Comm_From_Carrier01.Status.Y_Position, Z := Comm_From_Carrier01.Status.Z_Position, XTrack_X_Values := XTrack_X_Values, Transfergate => Transfergate_Car01); END_IF;

